LIN {X 0,Y 311.658,Z 464.201,A -85,B 0,C 180,E1 -15739.607,E2 -15739.607} C_VEL
LIN {X 0,Y 311.053,Z 468.336,A -85,B 0,C 180,E1 -15742.209,E2 -15742.209} C_VEL
LIN {X 0,Y 310.773,Z 471.242,A -85,B 0,C 180,E1 -15744.81,E2 -15744.81} C_VEL
LIN {X 0,Y 310.678,Z 472.99,A -85,B 0,C 180,E1 -15747.407,E2 -15747.407} C_VEL
LIN {X 0,Y 310.617,Z 473.6,A -85,B 0,C 180,E1 -15750,E2 -15750} C_VEL
LIN {X 0,Y 310.678,Z 473.032,A -85,B 0,C 180,E1 -15752.593,E2 -15752.593} C_VEL
LIN {X 0,Y 310.76,Z 471.342,A -85,B 0,C 180,E1 -15755.19,E2 -15755.19} C_VEL
LIN {X 0,Y 311.014,Z 468.49,A -85,B 0,C 180,E1 -15757.792,E2 -15757.792} C_VEL
LIN {X 0,Y 311.62,Z 464.406,A -85,B 0,C 180,E1 -15760.395,E2 -15760.395} C_VEL
LIN {X 0,Y 312.631,Z 458.992,A -85,B 0,C 180,E1 -15762.991,E2 -15762.991} C_VEL
LIN {X 0,Y 313.876,Z 452.096,A -85,B 0,C 180,E1 -15765.587,E2 -15765.587} C_VEL
LIN {X 0,Y 315.733,Z 443.488,A -85,B 0,C 180,E1 -15768.158,E2 -15768.158} C_VEL
LIN {X 0,Y 317.704,Z 434.339,A -85,B 0,C 180,E1 -15770.39,E2 -15770.39} C_VEL
LIN {X 0,Y 319.854,Z 424.962,A -85,B 0,C 180,E1 -15772.285,E2 -15772.285} C_VEL
LIN {X 0,Y 322.098,Z 413.952,A -85,B 0,C 180,E1 -15774.149,E2 -15774.149} C_VEL
LIN {X 0,Y 324.511,Z 401.832,A -85,B 0,C 180,E1 -15775.84,E2 -15775.84} C_VEL
LIN {X 0,Y 326.933,Z 388.524,A -85,B 0,C 180,E1 -15777.355,E2 -15777.355} C_VEL
LIN {X 0,Y 329.075,Z 375.209,A -85,B 0,C 180,E1 -15778.572,E2 -15778.572} C_VEL
LIN {X 0,Y 331.025,Z 360.086,A -85,B 0,C 180,E1 -15779.666,E2 -15779.666} C_VEL
LIN {X 0,Y 332.582,Z 345.03,A -85,B 0,C 180,E1 -15780.475,E2 -15780.475} C_VEL
LIN {X 0,Y 333.767,Z 329.274,A -85,B 0,C 180,E1 -15781.057,E2 -15781.057} C_VEL
LIN {X 0,Y 335.921,Z 270.181,A -85,B 0,C 180,E1 -15782.336,E2 -15782.336} C_VEL
LIN {X 0,Y 336.412,Z 254.41,A -85,B 0,C 180,E1 -15782.674,E2 -15782.674} C_VEL
LIN {X 0,Y 336.043,Z 248.619,A -85,B 0,C 180,E1 -15782.859,E2 -15782.859} C_VEL
LIN {X 0,Y 331.98,Z 229.992,A -85,B 0,C 180,E1 -15783.788,E2 -15783.788} C_VEL
LIN {X 0,Y 331.521,Z 224.208,A -85,B 0,C 180,E1 -15783.989,E2 -15783.989} C_VEL
LIN {X 0,Y 331.82,Z 212.788,A -85,B 0,C 180,E1 -15784.246,E2 -15784.246} C_VEL
LIN {X 0,Y 324.4,Z 195.968,A -85,B 0,C 180,E1 -15785.592,E2 -15785.592} C_VEL
LIN {X 0,Y 316.403,Z 180.051,A -85,B 0,C 180,E1 -15787.08,E2 -15787.08} C_VEL
LIN {X 0,Y 308.749,Z 166.539,A -85,B 0,C 180,E1 -15788.556,E2 -15788.556} C_VEL
LIN {X 0,Y 306.876,Z 163.029,A -85,B 0,C 180,E1 -15789.022,E2 -15789.022} C_VEL
LIN {X 0,Y 305.465,Z 158.467,A -85,B 0,C 180,E1 -15790.602,E2 -15790.602} C_VEL
LIN {X 0,Y 305.39,Z 158.081,A -85,B 0,C 180,E1 -15790.91,E2 -15790.91} C_VEL
LIN {X 0,Y 305.399,Z 158.043,A -85,B 0,C 180,E1 -15794.489,E2 -15794.489} C_VEL
LIN {X 0,Y 305.411,Z 158.038,A -85,B 0,C 180,E1 -15798.138,E2 -15798.138} C_VEL
LIN {X 0,Y 305.442,Z 158.029,A -85,B 0,C 180,E1 -15801.592,E2 -15801.592} C_VEL
LIN {X 0,Y 305.463,Z 158.048,A -85,B 0,C 180,E1 -15804.887,E2 -15804.887} C_VEL
LIN {X 0,Y 305.442,Z 158.001,A -85,B 0,C 180,E1 -15808.359,E2 -15808.359} C_VEL
LIN {X 0,Y 305.476,Z 158.046,A -85,B 0,C 180,E1 -15811.109,E2 -15811.109} C_VEL
LIN {X 0,Y 305.482,Z 158.044,A -85,B 0,C 180,E1 -15814.08,E2 -15814.08} C_VEL
LIN {X 0,Y 305.473,Z 158.052,A -85,B 0,C 180,E1 -15818.401,E2 -15818.401} C_VEL
LIN {X 0,Y 305.529,Z 158.052,A -85,B 0,C 180,E1 -15822.6,E2 -15822.6} C_VEL
LIN {X 0,Y 305.625,Z 158.019,A -85,B 0,C 180,E1 -15825.348,E2 -15825.348} C_VEL
LIN {X 0,Y 305.626,Z 158.037,A -85,B 0,C 180,E1 -15829.399,E2 -15829.399} C_VEL
LIN {X 0,Y 305.751,Z 158.004,A -85,B 0,C 180,E1 -15832.073,E2 -15832.073} C_VEL
LIN {X 0,Y 305.669,Z 158.033,A -85,B 0,C 180,E1 -15834.723,E2 -15834.723} C_VEL
LIN {X 0,Y 305.949,Z 157.982,A -85,B 0,C 180,E1 -15838.684,E2 -15838.684} C_VEL
LIN {X 0,Y 305.951,Z 157.995,A -85,B 0,C 180,E1 -15841.316,E2 -15841.316} C_VEL
LIN {X 0,Y 305.671,Z 158.022,A -85,B 0,C 180,E1 -15845.277,E2 -15845.277} C_VEL
LIN {X 0,Y 305.751,Z 158.016,A -85,B 0,C 180,E1 -15847.927,E2 -15847.927} C_VEL
LIN {X 0,Y 305.601,Z 158.043,A -85,B 0,C 180,E1 -15851.945,E2 -15851.945} C_VEL
LIN {X 0,Y 305.639,Z 158.019,A -85,B 0,C 180,E1 -15855.035,E2 -15855.035} C_VEL
LIN {X 0,Y 305.581,Z 158.045,A -85,B 0,C 180,E1 -15858.783,E2 -15858.783} C_VEL
LIN {X 0,Y 305.487,Z 158.055,A -85,B 0,C 180,E1 -15863.039,E2 -15863.039} C_VEL
LIN {X 0,Y 305.527,Z 158.035,A -85,B 0,C 180,E1 -15866.219,E2 -15866.219} C_VEL
LIN {X 0,Y 305.497,Z 158.054,A -85,B 0,C 180,E1 -15869.05,E2 -15869.05} C_VEL
LIN {X 0,Y 305.465,Z 158.001,A -85,B 0,C 180,E1 -15873.517,E2 -15873.517} C_VEL
LIN {X 0,Y 305.473,Z 158.06,A -85,B 0,C 180,E1 -15876.739,E2 -15876.739} C_VEL
LIN {X 0,Y 305.455,Z 158.021,A -85,B 0,C 180,E1 -15880.599,E2 -15880.599} C_VEL
LIN {X 0,Y 305.426,Z 158.066,A -85,B 0,C 180,E1 -15883.655,E2 -15883.655} C_VEL
LIN {X 0,Y 305.506,Z 158.163,A -85,B 0,C 180,E1 -15888.12,E2 -15888.12} C_VEL
LIN {X 0,Y 308.349,Z 167.712,A -85,B 0,C 180,E1 -15891.296,E2 -15891.296} C_VEL
LIN {X 0,Y 316.324,Z 182.462,A -85,B 0,C 180,E1 -15892.89,E2 -15892.89} C_VEL
LIN {X 0,Y 323.257,Z 196.28,A -85,B 0,C 180,E1 -15894.184,E2 -15894.184} C_VEL
LIN {X 0,Y 331.081,Z 213.937,A -85,B 0,C 180,E1 -15895.609,E2 -15895.609} C_VEL
LIN {X 0,Y 331.761,Z 218.64,A -85,B 0,C 180,E1 -15895.81,E2 -15895.81} C_VEL
LIN {X 0,Y 328.229,Z 318.553,A -85,B 0,C 180,E1 -15897.953,E2 -15897.953} C_VEL
LIN {X 0,Y 327.363,Z 337.959,A -85,B 0,C 180,E1 -15898.446,E2 -15898.446} C_VEL
LIN {X 0,Y 325.998,Z 353.359,A -85,B 0,C 180,E1 -15899.067,E2 -15899.067} C_VEL
LIN {X 0,Y 324.342,Z 367.08,A -85,B 0,C 180,E1 -15899.838,E2 -15899.838} C_VEL
LIN {X 0,Y 322.371,Z 381.795,A -85,B 0,C 180,E1 -15900.949,E2 -15900.949} C_VEL
LIN {X 0,Y 320.123,Z 394.944,A -85,B 0,C 180,E1 -15902.191,E2 -15902.191} C_VEL
LIN {X 0,Y 317.506,Z 408.093,A -85,B 0,C 180,E1 -15903.724,E2 -15903.724} C_VEL
LIN {X 0,Y 315.186,Z 419.121,A -85,B 0,C 180,E1 -15905.286,E2 -15905.286} C_VEL
LIN {X 0,Y 312.947,Z 429.414,A -85,B 0,C 180,E1 -15907.037,E2 -15907.037} C_VEL
LIN {X 0,Y 310.691,Z 439.64,A -85,B 0,C 180,E1 -15909.128,E2 -15909.128} C_VEL
LIN {X 0,Y 308.58,Z 448.862,A -85,B 0,C 180,E1 -15911.406,E2 -15911.406} C_VEL
LIN {X 0,Y 306.705,Z 457.543,A -85,B 0,C 180,E1 -15914.039,E2 -15914.039} C_VEL
LIN {X 0,Y 305.38,Z 464.508,A -85,B 0,C 180,E1 -15916.695,E2 -15916.695} C_VEL
LIN {X 0,Y 304.395,Z 469.982,A -85,B 0,C 180,E1 -15919.356,E2 -15919.356} C_VEL
LIN {X 0,Y 303.868,Z 474.121,A -85,B 0,C 180,E1 -15922.023,E2 -15922.023} C_VEL
LIN {X 0,Y 303.596,Z 477.021,A -85,B 0,C 180,E1 -15924.687,E2 -15924.687} C_VEL
LIN {X 0,Y 303.57,Z 478.751,A -85,B 0,C 180,E1 -15927.346,E2 -15927.346} C_VEL
LIN {X 0,Y 303.531,Z 479.341,A -85,B 0,C 180,E1 -15930,E2 -15930} C_VEL
LIN {X 0,Y 303.57,Z 478.741,A -85,B 0,C 180,E1 -15932.654,E2 -15932.654} C_VEL
LIN {X 0,Y 303.624,Z 476.802,A -85,B 0,C 180,E1 -15935.544,E2 -15935.544} C_VEL
LIN {X 0,Y 303.867,Z 474.09,A -85,B 0,C 180,E1 -15937.977,E2 -15937.977} C_VEL
LIN {X 0,Y 304.388,Z 469.945,A -85,B 0,C 180,E1 -15940.644,E2 -15940.644} C_VEL
LIN {X 0,Y 305.369,Z 464.455,A -85,B 0,C 180,E1 -15943.306,E2 -15943.306} C_VEL
LIN {X 0,Y 306.657,Z 457.468,A -85,B 0,C 180,E1 -15945.963,E2 -15945.963} C_VEL
LIN {X 0,Y 308.568,Z 448.775,A -85,B 0,C 180,E1 -15948.594,E2 -15948.594} C_VEL
LIN {X 0,Y 310.704,Z 439.539,A -85,B 0,C 180,E1 -15950.871,E2 -15950.871} C_VEL
LIN {X 0,Y 312.746,Z 429.81,A -85,B 0,C 180,E1 -15952.876,E2 -15952.876} C_VEL
LIN {X 0,Y 315.433,Z 417.964,A -85,B 0,C 180,E1 -15954.869,E2 -15954.869} C_VEL
LIN {X 0,Y 317.982,Z 405.536,A -85,B 0,C 180,E1 -15956.587,E2 -15956.587} C_VEL
LIN {X 0,Y 320.353,Z 393.309,A -85,B 0,C 180,E1 -15957.965,E2 -15957.965} C_VEL
LIN {X 0,Y 322.79,Z 378.654,A -85,B 0,C 180,E1 -15959.297,E2 -15959.297} C_VEL
LIN {X 0,Y 324.654,Z 364.495,A -85,B 0,C 180,E1 -15960.309,E2 -15960.309} C_VEL
LIN {X 0,Y 326.377,Z 349.088,A -85,B 0,C 180,E1 -15961.118,E2 -15961.118} C_VEL
LIN {X 0,Y 327.591,Z 333.851,A -85,B 0,C 180,E1 -15961.664,E2 -15961.664} C_VEL
LIN {X 0,Y 331.459,Z 224.627,A -85,B 0,C 180,E1 -15964.044,E2 -15964.044} C_VEL
LIN {X 0,Y 331.527,Z 216.912,A -85,B 0,C 180,E1 -15964.233,E2 -15964.233} C_VEL
LIN {X 0,Y 330.749,Z 213.239,A -85,B 0,C 180,E1 -15964.419,E2 -15964.419} C_VEL
LIN {X 0,Y 322.793,Z 195.303,A -85,B 0,C 180,E1 -15965.87,E2 -15965.87} C_VEL
LIN {X 0,Y 314.623,Z 179.237,A -85,B 0,C 180,E1 -15967.4,E2 -15967.4} C_VEL
LIN {X 0,Y 309.575,Z 170.227,A -85,B 0,C 180,E1 -15968.376,E2 -15968.376} C_VEL
LIN {X 0,Y 308.28,Z 167.558,A -85,B 0,C 180,E1 -15968.701,E2 -15968.701} C_VEL
LIN {X 0,Y 305.477,Z 158.164,A -85,B 0,C 180,E1 -15971.851,E2 -15971.851} C_VEL
LIN {X 0,Y 305.4,Z 158.054,A -85,B 0,C 180,E1 -15975.511,E2 -15975.511} C_VEL
LIN {X 0,Y 305.44,Z 158.034,A -85,B 0,C 180,E1 -15978.143,E2 -15978.143} C_VEL
LIN {X 0,Y 305.495,Z 158.041,A -85,B 0,C 180,E1 -15981.6,E2 -15981.6} C_VEL
LIN {X 0,Y 305.462,Z 158.025,A -85,B 0,C 180,E1 -15984.887,E2 -15984.887} C_VEL
LIN {X 0,Y 305.451,Z 158.011,A -85,B 0,C 180,E1 -15988.355,E2 -15988.355} C_VEL
LIN {X 0,Y 305.521,Z 158.053,A -85,B 0,C 180,E1 -15991.114,E2 -15991.114} C_VEL
LIN {X 0,Y 305.572,Z 158.029,A -85,B 0,C 180,E1 -15994.088,E2 -15994.088} C_VEL
LIN {X 0,Y 305.501,Z 158.039,A -85,B 0,C 180,E1 -15998.403,E2 -15998.403} C_VEL
LIN {X 0,Y 305.591,Z 158.044,A -85,B 0,C 180,E1 -16001.218,E2 -16001.218} C_VEL
LIN {X 0,Y 305.65,Z 158.021,A -85,B 0,C 180,E1 -16005.349,E2 -16005.349} C_VEL
LIN {X 0,Y 305.625,Z 158.022,A -85,B 0,C 180,E1 -16009.399,E2 -16009.399} C_VEL
LIN {X 0,Y 305.75,Z 158.016,A -85,B 0,C 180,E1 -16012.073,E2 -16012.073} C_VEL
LIN {X 0,Y 305.671,Z 158.022,A -85,B 0,C 180,E1 -16014.723,E2 -16014.723} C_VEL
LIN {X 0,Y 305.953,Z 157.994,A -85,B 0,C 180,E1 -16018.684,E2 -16018.684} C_VEL
LIN {X 0,Y 305.951,Z 157.982,A -85,B 0,C 180,E1 -16021.316,E2 -16021.316} C_VEL
LIN {X 0,Y 305.794,Z 158.012,A -85,B 0,C 180,E1 -16026.599,E2 -16026.599} C_VEL
LIN {X 0,Y 305.695,Z 158.012,A -85,B 0,C 180,E1 -16029.261,E2 -16029.261} C_VEL
LIN {X 0,Y 305.587,Z 158.031,A -85,B 0,C 180,E1 -16033.296,E2 -16033.296} C_VEL
LIN {X 0,Y 305.552,Z 158.039,A -85,B 0,C 180,E1 -16036.023,E2 -16036.023} C_VEL
LIN {X 0,Y 305.484,Z 158.038,A -85,B 0,C 180,E1 -16040.188,E2 -16040.188} C_VEL
LIN {X 0,Y 305.442,Z 158.048,A -85,B 0,C 180,E1 -16044.467,E2 -16044.467} C_VEL
LIN {X 0,Y 305.452,Z 158.061,A -85,B 0,C 180,E1 -16047.398,E2 -16047.398} C_VEL
LIN {X 0,Y 305.429,Z 158.02,A -85,B 0,C 180,E1 -16050.413,E2 -16050.413} C_VEL
LIN {X 0,Y 305.465,Z 158.017,A -85,B 0,C 180,E1 -16054.078,E2 -16054.078} C_VEL
LIN {X 0,Y 305.469,Z 158.062,A -85,B 0,C 180,E1 -16056.74,E2 -16056.74} C_VEL
LIN {X 0,Y 305.409,Z 158.019,A -85,B 0,C 180,E1 -16060.59,E2 -16060.59} C_VEL
LIN {X 0,Y 305.421,Z 158.066,A -85,B 0,C 180,E1 -16063.656,E2 -16063.656} C_VEL
LIN {X 0,Y 305.435,Z 158.05,A -85,B 0,C 180,E1 -16067.419,E2 -16067.419} C_VEL
LIN {X 0,Y 305.42,Z 158.229,A -85,B 0,C 180,E1 -16069.408,E2 -16069.408} C_VEL
LIN {X 0,Y 306.99,Z 163.275,A -85,B 0,C 180,E1 -16071.167,E2 -16071.167} C_VEL
LIN {X 0,Y 314.485,Z 176.51,A -85,B 0,C 180,E1 -16072.68,E2 -16072.68} C_VEL
LIN {X 0,Y 322.078,Z 191.253,A -85,B 0,C 180,E1 -16074.106,E2 -16074.106} C_VEL
LIN {X 0,Y 329.975,Z 208.394,A -85,B 0,C 180,E1 -16075.54,E2 -16075.54} C_VEL
LIN {X 0,Y 331.749,Z 212.616,A -85,B 0,C 180,E1 -16075.859,E2 -16075.859} C_VEL
LIN {X 0,Y 328.421,Z 312.293,A -85,B 0,C 180,E1 -16078.019,E2 -16078.019} C_VEL
LIN {X 0,Y 327.446,Z 332.079,A -85,B 0,C 180,E1 -16078.5,E2 -16078.5} C_VEL
LIN {X 0,Y 326.21,Z 347.317,A -85,B 0,C 180,E1 -16079.112,E2 -16079.112} C_VEL
LIN {X 0,Y 324.689,Z 361.386,A -85,B 0,C 180,E1 -16079.909,E2 -16079.909} C_VEL
LIN {X 0,Y 322.785,Z 375.372,A -85,B 0,C 180,E1 -16080.946,E2 -16080.946} C_VEL
LIN {X 0,Y 320.494,Z 389.08,A -85,B 0,C 180,E1 -16082.226,E2 -16082.226} C_VEL
LIN {X 0,Y 318.241,Z 401.138,A -85,B 0,C 180,E1 -16083.613,E2 -16083.613} C_VEL
LIN {X 0,Y 315.637,Z 413.38,A -85,B 0,C 180,E1 -16085.324,E2 -16085.324} C_VEL
LIN {X 0,Y 313.181,Z 425.143,A -85,B 0,C 180,E1 -16087.354,E2 -16087.354} C_VEL
LIN {X 0,Y 310.79,Z 435.369,A -85,B 0,C 180,E1 -16089.482,E2 -16089.482} C_VEL
LIN {X 0,Y 308.73,Z 444.365,A -85,B 0,C 180,E1 -16091.759,E2 -16091.759} C_VEL
LIN {X 0,Y 306.988,Z 451.821,A -85,B 0,C 180,E1 -16094.055,E2 -16094.055} C_VEL
LIN {X 0,Y 305.697,Z 458.79,A -85,B 0,C 180,E1 -16096.709,E2 -16096.709} C_VEL
LIN {X 0,Y 304.634,Z 464.268,A -85,B 0,C 180,E1 -16099.364,E2 -16099.364} C_VEL
LIN {X 0,Y 304.006,Z 468.404,A -85,B 0,C 180,E1 -16102.027,E2 -16102.027} C_VEL
LIN {X 0,Y 303.686,Z 471.309,A -85,B 0,C 180,E1 -16104.689,E2 -16104.689} C_VEL
LIN {X 0,Y 303.604,Z 473.056,A -85,B 0,C 180,E1 -16107.346,E2 -16107.346} C_VEL
LIN {X 0,Y 303.533,Z 473.666,A -85,B 0,C 180,E1 -16110,E2 -16110} C_VEL
LIN {X 0,Y 303.603,Z 473.098,A -85,B 0,C 180,E1 -16112.654,E2 -16112.654} C_VEL
LIN {X 0,Y 303.73,Z 471.045,A -85,B 0,C 180,E1 -16115.744,E2 -16115.744} C_VEL
LIN {X 0,Y 303.976,Z 468.555,A -85,B 0,C 180,E1 -16117.974,E2 -16117.974} C_VEL
LIN {X 0,Y 304.602,Z 464.471,A -85,B 0,C 180,E1 -16120.637,E2 -16120.637} C_VEL
LIN {X 0,Y 305.657,Z 459.057,A -85,B 0,C 180,E1 -16123.293,E2 -16123.293} C_VEL
LIN {X 0,Y 306.989,Z 452.161,A -85,B 0,C 180,E1 -16125.945,E2 -16125.945} C_VEL
LIN {X 0,Y 308.94,Z 443.553,A -85,B 0,C 180,E1 -16128.571,E2 -16128.571} C_VEL
LIN {X 0,Y 311.026,Z 434.403,A -85,B 0,C 180,E1 -16130.848,E2 -16130.848} C_VEL
LIN {X 0,Y 313.174,Z 425.31,A -85,B 0,C 180,E1 -16132.726,E2 -16132.726} C_VEL
LIN {X 0,Y 315.592,Z 414.015,A -85,B 0,C 180,E1 -16134.68,E2 -16134.68} C_VEL
LIN {X 0,Y 318.088,Z 401.895,A -85,B 0,C 180,E1 -16136.401,E2 -16136.401} C_VEL
LIN {X 0,Y 320.625,Z 388.586,A -85,B 0,C 180,E1 -16137.939,E2 -16137.939} C_VEL
LIN {X 0,Y 322.811,Z 375.586,A -85,B 0,C 180,E1 -16139.147,E2 -16139.147} C_VEL
LIN {X 0,Y 324.731,Z 361.274,A -85,B 0,C 180,E1 -16140.211,E2 -16140.211} C_VEL
LIN {X 0,Y 326.352,Z 346.609,A -85,B 0,C 180,E1 -16141.031,E2 -16141.031} C_VEL
LIN {X 0,Y 327.575,Z 331.603,A -85,B 0,C 180,E1 -16141.621,E2 -16141.621} C_VEL
LIN {X 0,Y 328.533,Z 309.767,A -85,B 0,C 180,E1 -16142.149,E2 -16142.149} C_VEL
LIN {X 0,Y 331.521,Z 224.208,A -85,B 0,C 180,E1 -16143.989,E2 -16143.989} C_VEL
LIN {X 0,Y 330.934,Z 220.467,A -85,B 0,C 180,E1 -16144.153,E2 -16144.153} C_VEL
LIN {X 0,Y 329.477,Z 217.097,A -85,B 0,C 180,E1 -16144.413,E2 -16144.413} C_VEL
LIN {X 0,Y 322.573,Z 206.994,A -85,B 0,C 180,E1 -16145.529,E2 -16145.529} C_VEL
LIN {X 0,Y 314.231,Z 189.381,A -85,B 0,C 180,E1 -16147.118,E2 -16147.118} C_VEL
LIN {X 0,Y 306.471,Z 175.095,A -85,B 0,C 180,E1 -16148.644,E2 -16148.644} C_VEL
LIN {X 0,Y 299.708,Z 163.412,A -85,B 0,C 180,E1 -16150.089,E2 -16150.089} C_VEL
LIN {X 0,Y 298.405,Z 159.201,A -85,B 0,C 180,E1 -16151.593,E2 -16151.593} C_VEL
LIN {X 0,Y 298.37,Z 158.924,A -85,B 0,C 180,E1 -16153.097,E2 -16153.097} C_VEL
LIN {X 0,Y 298.371,Z 158.944,A -85,B 0,C 180,E1 -16156.915,E2 -16156.915} C_VEL
LIN {X 0,Y 298.352,Z 158.902,A -85,B 0,C 180,E1 -16161.019,E2 -16161.019} C_VEL
LIN {X 0,Y 298.406,Z 158.942,A -85,B 0,C 180,E1 -16163.928,E2 -16163.928} C_VEL
LIN {X 0,Y 298.393,Z 158.88,A -85,B 0,C 180,E1 -16167.199,E2 -16167.199} C_VEL
LIN {X 0,Y 298.402,Z 158.917,A -85,B 0,C 180,E1 -16170.625,E2 -16170.625} C_VEL
LIN {X 0,Y 298.416,Z 158.92,A -85,B 0,C 180,E1 -16174.918,E2 -16174.918} C_VEL
LIN {X 0,Y 298.401,Z 158.939,A -85,B 0,C 180,E1 -16177.862,E2 -16177.862} C_VEL
LIN {X 0,Y 298.465,Z 158.914,A -85,B 0,C 180,E1 -16180.752,E2 -16180.752} C_VEL
LIN {X 0,Y 298.587,Z 158.897,A -85,B 0,C 180,E1 -16184.994,E2 -16184.994} C_VEL
LIN {X 0,Y 298.585,Z 158.917,A -85,B 0,C 180,E1 -16189.146,E2 -16189.146} C_VEL
LIN {X 0,Y 298.702,Z 158.88,A -85,B 0,C 180,E1 -16191.884,E2 -16191.884} C_VEL
LIN {X 0,Y 298.639,Z 158.909,A -85,B 0,C 180,E1 -16194.598,E2 -16194.598} C_VEL
LIN {X 0,Y 298.916,Z 158.857,A -85,B 0,C 180,E1 -16198.653,E2 -16198.653} C_VEL
LIN {X 0,Y 298.918,Z 158.87,A -85,B 0,C 180,E1 -16201.347,E2 -16201.347} C_VEL
LIN {X 0,Y 298.64,Z 158.899,A -85,B 0,C 180,E1 -16205.401,E2 -16205.401} C_VEL
LIN {X 0,Y 298.702,Z 158.892,A -85,B 0,C 180,E1 -16208.115,E2 -16208.115} C_VEL
LIN {X 0,Y 298.553,Z 158.92,A -85,B 0,C 180,E1 -16212.231,E2 -16212.231} C_VEL
LIN {X 0,Y 298.607,Z 158.894,A -85,B 0,C 180,E1 -16215.209,E2 -16215.209} C_VEL
LIN {X 0,Y 298.527,Z 158.919,A -85,B 0,C 180,E1 -16219.244,E2 -16219.244} C_VEL
LIN {X 0,Y 298.43,Z 158.936,A -85,B 0,C 180,E1 -16223.6,E2 -16223.6} C_VEL
LIN {X 0,Y 298.487,Z 158.912,A -85,B 0,C 180,E1 -16226.574,E2 -16226.574} C_VEL
LIN {X 0,Y 298.422,Z 158.927,A -85,B 0,C 180,E1 -16229.641,E2 -16229.641} C_VEL
LIN {X 0,Y 298.396,Z 158.878,A -85,B 0,C 180,E1 -16232.8,E2 -16232.8} C_VEL
LIN {X 0,Y 298.445,Z 158.936,A -85,B 0,C 180,E1 -16236.807,E2 -16236.807} C_VEL
LIN {X 0,Y 298.387,Z 158.903,A -85,B 0,C 180,E1 -16241.087,E2 -16241.087} C_VEL
LIN {X 0,Y 298.399,Z 158.939,A -85,B 0,C 180,E1 -16243.103,E2 -16243.103} C_VEL
LIN {X 0,Y 298.447,Z 159.078,A -85,B 0,C 180,E1 -16247.211,E2 -16247.211} C_VEL
LIN {X 0,Y 301.023,Z 167.6,A -85,B 0,C 180,E1 -16250.165,E2 -16250.165} C_VEL
LIN {X 0,Y 308.862,Z 181.664,A -85,B 0,C 180,E1 -16251.814,E2 -16251.814} C_VEL
LIN {X 0,Y 316.721,Z 197.093,A -85,B 0,C 180,E1 -16253.35,E2 -16253.35} C_VEL
LIN {X 0,Y 324.301,Z 213.884,A -85,B 0,C 180,E1 -16254.785,E2 -16254.785} C_VEL
LIN {X 0,Y 325.615,Z 217.399,A -85,B 0,C 180,E1 -16255.041,E2 -16255.041} C_VEL
LIN {X 0,Y 325.839,Z 220.532,A -85,B 0,C 180,E1 -16255.151,E2 -16255.151} C_VEL
LIN {X 0,Y 321.658,Z 333.25,A -85,B 0,C 180,E1 -16257.635,E2 -16257.635} C_VEL
LIN {X 0,Y 320.42,Z 348.658,A -85,B 0,C 180,E1 -16258.19,E2 -16258.19} C_VEL
LIN {X 0,Y 318.687,Z 363.552,A -85,B 0,C 180,E1 -16258.97,E2 -16258.97} C_VEL
LIN {X 0,Y 316.849,Z 377.218,A -85,B 0,C 180,E1 -16259.943,E2 -16259.943} C_VEL
LIN {X 0,Y 314.643,Z 390.368,A -85,B 0,C 180,E1 -16261.117,E2 -16261.117} C_VEL
LIN {X 0,Y 312.16,Z 403.064,A -85,B 0,C 180,E1 -16262.513,E2 -16262.513} C_VEL
LIN {X 0,Y 309.452,Z 415.905,A -85,B 0,C 180,E1 -16264.256,E2 -16264.256} C_VEL
LIN {X 0,Y 307.023,Z 426.604,A -85,B 0,C 180,E1 -16266.016,E2 -16266.016} C_VEL
LIN {X 0,Y 304.739,Z 436.601,A -85,B 0,C 180,E1 -16267.99,E2 -16267.99} C_VEL
LIN {X 0,Y 302.377,Z 446.329,A -85,B 0,C 180,E1 -16270.305,E2 -16270.305} C_VEL
LIN {X 0,Y 300.448,Z 454.446,A -85,B 0,C 180,E1 -16272.648,E2 -16272.648} C_VEL
LIN {X 0,Y 299.056,Z 461.158,A -85,B 0,C 180,E1 -16275.018,E2 -16275.018} C_VEL
LIN {X 0,Y 297.799,Z 467.354,A -85,B 0,C 180,E1 -16277.737,E2 -16277.737} C_VEL
LIN {X 0,Y 297.052,Z 472.145,A -85,B 0,C 180,E1 -16280.467,E2 -16280.467} C_VEL
LIN {X 0,Y 296.642,Z 475.655,A -85,B 0,C 180,E1 -16283.197,E2 -16283.197} C_VEL
LIN {X 0,Y 296.468,Z 477.963,A -85,B 0,C 180,E1 -16285.922,E2 -16285.922} C_VEL
LIN {X 0,Y 296.444,Z 479.123,A -85,B 0,C 180,E1 -16288.641,E2 -16288.641} C_VEL
LIN {X 0,Y 296.444,Z 479.119,A -85,B 0,C 180,E1 -16291.358,E2 -16291.358} C_VEL
LIN {X 0,Y 296.469,Z 477.946,A -85,B 0,C 180,E1 -16294.078,E2 -16294.078} C_VEL
LIN {X 0,Y 296.642,Z 475.626,A -85,B 0,C 180,E1 -16296.803,E2 -16296.803} C_VEL
LIN {X 0,Y 297.048,Z 472.11,A -85,B 0,C 180,E1 -16299.533,E2 -16299.533} C_VEL
LIN {X 0,Y 297.795,Z 467.309,A -85,B 0,C 180,E1 -16302.263,E2 -16302.263} C_VEL
LIN {X 0,Y 299.009,Z 461.091,A -85,B 0,C 180,E1 -16304.984,E2 -16304.984} C_VEL
LIN {X 0,Y 300.715,Z 453.283,A -85,B 0,C 180,E1 -16307.687,E2 -16307.687} C_VEL
LIN {X 0,Y 302.622,Z 444.979,A -85,B 0,C 180,E1 -16310.032,E2 -16310.032} C_VEL
LIN {X 0,Y 305.081,Z 434.973,A -85,B 0,C 180,E1 -16312.34,E2 -16312.34} C_VEL
LIN {X 0,Y 306.924,Z 426.703,A -85,B 0,C 180,E1 -16313.946,E2 -16313.946} C_VEL
LIN {X 0,Y 309.459,Z 415.754,A -85,B 0,C 180,E1 -16315.743,E2 -16315.743} C_VEL
LIN {X 0,Y 311.903,Z 404.172,A -85,B 0,C 180,E1 -16317.329,E2 -16317.329} C_VEL
LIN {X 0,Y 314.338,Z 391.709,A -85,B 0,C 180,E1 -16318.731,E2 -16318.731} C_VEL
LIN {X 0,Y 316.759,Z 377.497,A -85,B 0,C 180,E1 -16320.012,E2 -16320.012} C_VEL
LIN {X 0,Y 318.667,Z 363.166,A -85,B 0,C 180,E1 -16321.032,E2 -16321.032} C_VEL
LIN {X 0,Y 320.406,Z 348.118,A -85,B 0,C 180,E1 -16321.811,E2 -16321.811} C_VEL
LIN {X 0,Y 321.585,Z 333.77,A -85,B 0,C 180,E1 -16322.327,E2 -16322.327} C_VEL
LIN {X 0,Y 325.684,Z 222.129,A -85,B 0,C 180,E1 -16324.796,E2 -16324.796} C_VEL
LIN {X 0,Y 325.534,Z 217.472,A -85,B 0,C 180,E1 -16324.937,E2 -16324.937} C_VEL
LIN {X 0,Y 323.681,Z 212.486,A -85,B 0,C 180,E1 -16325.298,E2 -16325.298} C_VEL
LIN {X 0,Y 315.367,Z 194.343,A -85,B 0,C 180,E1 -16326.875,E2 -16326.875} C_VEL
LIN {X 0,Y 307.59,Z 179.407,A -85,B 0,C 180,E1 -16328.4,E2 -16328.4} C_VEL
LIN {X 0,Y 301.013,Z 167.567,A -85,B 0,C 180,E1 -16329.8,E2 -16329.8} C_VEL
LIN {X 0,Y 298.452,Z 159.06,A -85,B 0,C 180,E1 -16332.756,E2 -16332.756} C_VEL
LIN {X 0,Y 298.403,Z 158.936,A -85,B 0,C 180,E1 -16336.921,E2 -16336.921} C_VEL
LIN {X 0,Y 298.415,Z 158.909,A -85,B 0,C 180,E1 -16341.004,E2 -16341.004} C_VEL
LIN {X 0,Y 298.432,Z 158.924,A -85,B 0,C 180,E1 -16343.932,E2 -16343.932} C_VEL
LIN {X 0,Y 298.395,Z 158.883,A -85,B 0,C 180,E1 -16347.984,E2 -16347.984} C_VEL
LIN {X 0,Y 298.464,Z 158.931,A -85,B 0,C 180,E1 -16351.905,E2 -16351.905} C_VEL
LIN {X 0,Y 298.487,Z 158.918,A -85,B 0,C 180,E1 -16354.924,E2 -16354.924} C_VEL
LIN {X 0,Y 298.45,Z 158.915,A -85,B 0,C 180,E1 -16359.315,E2 -16359.315} C_VEL
LIN {X 0,Y 298.539,Z 158.922,A -85,B 0,C 180,E1 -16362.18,E2 -16362.18} C_VEL
LIN {X 0,Y 298.594,Z 158.896,A -85,B 0,C 180,E1 -16364.995,E2 -16364.995} C_VEL
LIN {X 0,Y 298.584,Z 158.902,A -85,B 0,C 180,E1 -16369.146,E2 -16369.146} C_VEL
LIN {X 0,Y 298.701,Z 158.892,A -85,B 0,C 180,E1 -16371.885,E2 -16371.885} C_VEL
LIN {X 0,Y 298.64,Z 158.899,A -85,B 0,C 180,E1 -16374.599,E2 -16374.599} C_VEL
LIN {X 0,Y 298.92,Z 158.869,A -85,B 0,C 180,E1 -16378.653,E2 -16378.653} C_VEL
LIN {X 0,Y 298.917,Z 158.857,A -85,B 0,C 180,E1 -16381.347,E2 -16381.347} C_VEL
LIN {X 0,Y 298.742,Z 158.889,A -85,B 0,C 180,E1 -16386.755,E2 -16386.755} C_VEL
LIN {X 0,Y 298.626,Z 158.894,A -85,B 0,C 180,E1 -16389.482,E2 -16389.482} C_VEL
LIN {X 0,Y 298.546,Z 158.904,A -85,B 0,C 180,E1 -16393.616,E2 -16393.616} C_VEL
LIN {X 0,Y 298.485,Z 158.924,A -85,B 0,C 180,E1 -16396.412,E2 -16396.412} C_VEL
LIN {X 0,Y 298.443,Z 158.916,A -85,B 0,C 180,E1 -16399.617,E2 -16399.617} C_VEL
LIN {X 0,Y 298.383,Z 158.936,A -85,B 0,C 180,E1 -16403.604,E2 -16403.604} C_VEL
LIN {X 0,Y 298.403,Z 158.932,A -85,B 0,C 180,E1 -16406.583,E2 -16406.583} C_VEL
LIN {X 0,Y 298.393,Z 158.914,A -85,B 0,C 180,E1 -16409.644,E2 -16409.644} C_VEL
LIN {X 0,Y 298.393,Z 158.878,A -85,B 0,C 180,E1 -16412.801,E2 -16412.801} C_VEL
LIN {X 0,Y 298.441,Z 158.936,A -85,B 0,C 180,E1 -16416.806,E2 -16416.806} C_VEL
LIN {X 0,Y 298.347,Z 158.904,A -85,B 0,C 180,E1 -16421.268,E2 -16421.268} C_VEL
LIN {X 0,Y 298.355,Z 158.925,A -85,B 0,C 180,E1 -16425.035,E2 -16425.035} C_VEL
LIN {X 0,Y 298.384,Z 159.148,A -85,B 0,C 180,E1 -16428.513,E2 -16428.513} C_VEL
LIN {X 0,Y 299.702,Z 163.418,A -85,B 0,C 180,E1 -16430.041,E2 -16430.041} C_VEL
LIN {X 0,Y 307.751,Z 177.282,A -85,B 0,C 180,E1 -16431.738,E2 -16431.738} C_VEL
LIN {X 0,Y 315.801,Z 192.661,A -85,B 0,C 180,E1 -16433.313,E2 -16433.313} C_VEL
LIN {X 0,Y 322.916,Z 207.888,A -85,B 0,C 180,E1 -16434.659,E2 -16434.659} C_VEL
LIN {X 0,Y 325.822,Z 214.611,A -85,B 0,C 180,E1 -16435.199,E2 -16435.199} C_VEL
LIN {X 0,Y 322.71,Z 303.444,A -85,B 0,C 180,E1 -16437.152,E2 -16437.152} C_VEL
LIN {X 0,Y 321.636,Z 329.879,A -85,B 0,C 180,E1 -16437.772,E2 -16437.772} C_VEL
LIN {X 0,Y 320.424,Z 344.728,A -85,B 0,C 180,E1 -16438.33,E2 -16438.33} C_VEL
LIN {X 0,Y 318.745,Z 359.891,A -85,B 0,C 180,E1 -16439.16,E2 -16439.16} C_VEL
LIN {X 0,Y 316.764,Z 374.379,A -85,B 0,C 180,E1 -16440.228,E2 -16440.228} C_VEL
LIN {X 0,Y 314.51,Z 387.721,A -85,B 0,C 180,E1 -16441.468,E2 -16441.468} C_VEL
LIN {X 0,Y 311.858,Z 401.208,A -85,B 0,C 180,E1 -16443.029,E2 -16443.029} C_VEL
LIN {X 0,Y 309.172,Z 413.45,A -85,B 0,C 180,E1 -16444.772,E2 -16444.772} C_VEL
LIN {X 0,Y 306.702,Z 424.754,A -85,B 0,C 180,E1 -16446.748,E2 -16446.748} C_VEL
LIN {X 0,Y 304.099,Z 435.438,A -85,B 0,C 180,E1 -16449.009,E2 -16449.009} C_VEL
LIN {X 0,Y 301.961,Z 444.434,A -85,B 0,C 180,E1 -16451.336,E2 -16451.336} C_VEL
LIN {X 0,Y 300.012,Z 452.349,A -85,B 0,C 180,E1 -16453.833,E2 -16453.833} C_VEL
LIN {X 0,Y 298.741,Z 458.858,A -85,B 0,C 180,E1 -16456.393,E2 -16456.393} C_VEL
LIN {X 0,Y 297.621,Z 464.336,A -85,B 0,C 180,E1 -16459.111,E2 -16459.111} C_VEL
LIN {X 0,Y 296.951,Z 468.471,A -85,B 0,C 180,E1 -16461.836,E2 -16461.836} C_VEL
LIN {X 0,Y 296.621,Z 471.376,A -85,B 0,C 180,E1 -16464.562,E2 -16464.562} C_VEL
LIN {X 0,Y 296.531,Z 473.122,A -85,B 0,C 180,E1 -16467.283,E2 -16467.283} C_VEL
LIN {X 0,Y 296.452,Z 473.732,A -85,B 0,C 180,E1 -16470,E2 -16470} C_VEL
LIN {X 0,Y 296.53,Z 473.164,A -85,B 0,C 180,E1 -16472.717,E2 -16472.717} C_VEL
LIN {X 0,Y 296.631,Z 471.279,A -85,B 0,C 180,E1 -16475.676,E2 -16475.676} C_VEL
LIN {X 0,Y 296.928,Z 468.621,A -85,B 0,C 180,E1 -16478.165,E2 -16478.165} C_VEL
LIN {X 0,Y 297.594,Z 464.537,A -85,B 0,C 180,E1 -16480.89,E2 -16480.89} C_VEL
LIN {X 0,Y 298.699,Z 459.123,A -85,B 0,C 180,E1 -16483.609,E2 -16483.609} C_VEL
LIN {X 0,Y 300.118,Z 452.226,A -85,B 0,C 180,E1 -16486.321,E2 -16486.321} C_VEL
LIN {X 0,Y 302.17,Z 443.618,A -85,B 0,C 180,E1 -16489.003,E2 -16489.003} C_VEL
LIN {X 0,Y 304.356,Z 434.468,A -85,B 0,C 180,E1 -16491.327,E2 -16491.327} C_VEL
LIN {X 0,Y 306.521,Z 425.637,A -85,B 0,C 180,E1 -16493.19,E2 -16493.19} C_VEL
LIN {X 0,Y 309.138,Z 414.079,A -85,B 0,C 180,E1 -16495.231,E2 -16495.231} C_VEL
LIN {X 0,Y 311.728,Z 401.957,A -85,B 0,C 180,E1 -16496.983,E2 -16496.983} C_VEL
LIN {X 0,Y 314.362,Z 388.648,A -85,B 0,C 180,E1 -16498.546,E2 -16498.546} C_VEL
LIN {X 0,Y 316.717,Z 375.07,A -85,B 0,C 180,E1 -16499.824,E2 -16499.824} C_VEL
LIN {X 0,Y 318.739,Z 360.204,A -85,B 0,C 180,E1 -16500.933,E2 -16500.933} C_VEL
LIN {X 0,Y 320.431,Z 345.142,A -85,B 0,C 180,E1 -16501.762,E2 -16501.762} C_VEL
LIN {X 0,Y 321.691,Z 329.375,A -85,B 0,C 180,E1 -16502.361,E2 -16502.361} C_VEL
LIN {X 0,Y 324.144,Z 267.714,A -85,B 0,C 180,E1 -16503.73,E2 -16503.73} C_VEL
LIN {X 0,Y 325.898,Z 214.764,A -85,B 0,C 180,E1 -16504.907,E2 -16504.907} C_VEL
LIN {X 0,Y 322.573,Z 206.994,A -85,B 0,C 180,E1 -16505.529,E2 -16505.529} C_VEL
LIN {X 0,Y 318.53,Z 201.352,A -85,B 0,C 180,E1 -16506.205,E2 -16506.205} C_VEL
LIN {X 0,Y 309.29,Z 191.562,A -85,B 0,C 180,E1 -16507.752,E2 -16507.752} C_VEL
LIN {X 0,Y 305.39,Z 185.929,A -85,B 0,C 180,E1 -16508.487,E2 -16508.487} C_VEL
LIN {X 0,Y 299.104,Z 174.784,A -85,B 0,C 180,E1 -16509.793,E2 -16509.793} C_VEL
LIN {X 0,Y 292.435,Z 163.633,A -85,B 0,C 180,E1 -16511.282,E2 -16511.282} C_VEL
LIN {X 0,Y 291.354,Z 159.981,A -85,B 0,C 180,E1 -16512.612,E2 -16512.612} C_VEL
LIN {X 0,Y 291.29,Z 159.826,A -85,B 0,C 180,E1 -16516.37,E2 -16516.37} C_VEL
LIN {X 0,Y 291.311,Z 159.774,A -85,B 0,C 180,E1 -16520.535,E2 -16520.535} C_VEL
LIN {X 0,Y 291.397,Z 159.806,A -85,B 0,C 180,E1 -16522.918,E2 -16522.918} C_VEL
LIN {X 0,Y 291.345,Z 159.768,A -85,B 0,C 180,E1 -16526.301,E2 -16526.301} C_VEL
LIN {X 0,Y 291.365,Z 159.781,A -85,B 0,C 180,E1 -16530.268,E2 -16530.268} C_VEL
LIN {X 0,Y 291.344,Z 159.802,A -85,B 0,C 180,E1 -16534.265,E2 -16534.265} C_VEL
LIN {X 0,Y 291.354,Z 159.817,A -85,B 0,C 180,E1 -16537.297,E2 -16537.297} C_VEL
LIN {X 0,Y 291.391,Z 159.793,A -85,B 0,C 180,E1 -16540.265,E2 -16540.265} C_VEL
LIN {X 0,Y 291.499,Z 159.782,A -85,B 0,C 180,E1 -16544.666,E2 -16544.666} C_VEL
LIN {X 0,Y 291.531,Z 159.795,A -85,B 0,C 180,E1 -16548.88,E2 -16548.88} C_VEL
LIN {X 0,Y 291.655,Z 159.757,A -85,B 0,C 180,E1 -16551.687,E2 -16551.687} C_VEL
LIN {X 0,Y 291.608,Z 159.785,A -85,B 0,C 180,E1 -16554.468,E2 -16554.468} C_VEL
LIN {X 0,Y 291.882,Z 159.732,A -85,B 0,C 180,E1 -16558.62,E2 -16558.62} C_VEL
LIN {X 0,Y 291.885,Z 159.745,A -85,B 0,C 180,E1 -16561.38,E2 -16561.38} C_VEL
LIN {X 0,Y 291.693,Z 159.775,A -85,B 0,C 180,E1 -16566.919,E2 -16566.919} C_VEL
LIN {X 0,Y 291.57,Z 159.767,A -85,B 0,C 180,E1 -16569.714,E2 -16569.714} C_VEL
LIN {X 0,Y 291.524,Z 159.788,A -85,B 0,C 180,E1 -16573.95,E2 -16573.95} C_VEL
LIN {X 0,Y 291.488,Z 159.789,A -85,B 0,C 180,E1 -16576.818,E2 -16576.818} C_VEL
LIN {X 0,Y 291.452,Z 159.793,A -85,B 0,C 180,E1 -16579.875,E2 -16579.875} C_VEL
LIN {X 0,Y 291.384,Z 159.813,A -85,B 0,C 180,E1 -16584.207,E2 -16584.207} C_VEL
LIN {X 0,Y 291.422,Z 159.799,A -85,B 0,C 180,E1 -16587.271,E2 -16587.271} C_VEL
LIN {X 0,Y 291.338,Z 159.79,A -85,B 0,C 180,E1 -16590.437,E2 -16590.437} C_VEL
LIN {X 0,Y 291.345,Z 159.758,A -85,B 0,C 180,E1 -16593.698,E2 -16593.698} C_VEL
LIN {X 0,Y 291.373,Z 159.816,A -85,B 0,C 180,E1 -16597.253,E2 -16597.253} C_VEL
LIN {X 0,Y 291.332,Z 159.778,A -85,B 0,C 180,E1 -16600.642,E2 -16600.642} C_VEL
LIN {X 0,Y 291.291,Z 159.81,A -85,B 0,C 180,E1 -16604.402,E2 -16604.402} C_VEL
LIN {X 0,Y 291.346,Z 160.025,A -85,B 0,C 180,E1 -16606.248,E2 -16606.248} C_VEL
LIN {X 0,Y 293.68,Z 167.509,A -85,B 0,C 180,E1 -16608.958,E2 -16608.958} C_VEL
LIN {X 0,Y 301.764,Z 181.567,A -85,B 0,C 180,E1 -16610.745,E2 -16610.745} C_VEL
LIN {X 0,Y 311.24,Z 199.841,A -85,B 0,C 180,E1 -16612.675,E2 -16612.675} C_VEL
LIN {X 0,Y 319.896,Z 219.428,A -85,B 0,C 180,E1 -16614.378,E2 -16614.378} C_VEL
LIN {X 0,Y 319.698,Z 229.719,A -85,B 0,C 180,E1 -16614.63,E2 -16614.63} C_VEL
LIN {X 0,Y 315.685,Z 333.201,A -85,B 0,C 180,E1 -16616.945,E2 -16616.945} C_VEL
LIN {X 0,Y 314.418,Z 348.603,A -85,B 0,C 180,E1 -16617.51,E2 -16617.51} C_VEL
LIN {X 0,Y 312.638,Z 363.493,A -85,B 0,C 180,E1 -16618.3,E2 -16618.3} C_VEL
LIN {X 0,Y 310.592,Z 377.988,A -85,B 0,C 180,E1 -16619.352,E2 -16619.352} C_VEL
LIN {X 0,Y 308.157,Z 391.889,A -85,B 0,C 180,E1 -16620.637,E2 -16620.637} C_VEL
LIN {X 0,Y 305.307,Z 405.584,A -85,B 0,C 180,E1 -16622.216,E2 -16622.216} C_VEL
LIN {X 0,Y 302.51,Z 417.982,A -85,B 0,C 180,E1 -16623.991,E2 -16623.991} C_VEL
LIN {X 0,Y 299.97,Z 428.732,A -85,B 0,C 180,E1 -16625.868,E2 -16625.868} C_VEL
LIN {X 0,Y 297.74,Z 438.024,A -85,B 0,C 180,E1 -16627.81,E2 -16627.81} C_VEL
LIN {X 0,Y 295.324,Z 447.498,A -85,B 0,C 180,E1 -16630.177,E2 -16630.177} C_VEL
LIN {X 0,Y 293.357,Z 455.391,A -85,B 0,C 180,E1 -16632.574,E2 -16632.574} C_VEL
LIN {X 0,Y 291.754,Z 462.76,A -85,B 0,C 180,E1 -16635.349,E2 -16635.349} C_VEL
LIN {X 0,Y 290.55,Z 468.604,A -85,B 0,C 180,E1 -16638.135,E2 -16638.135} C_VEL
LIN {X 0,Y 290.015,Z 472.079,A -85,B 0,C 180,E1 -16640.233,E2 -16640.233} C_VEL
LIN {X 0,Y 289.566,Z 475.589,A -85,B 0,C 180,E1 -16643.03,E2 -16643.03} C_VEL
LIN {X 0,Y 289.373,Z 477.897,A -85,B 0,C 180,E1 -16645.822,E2 -16645.822} C_VEL
LIN {X 0,Y 289.368,Z 479.056,A -85,B 0,C 180,E1 -16648.608,E2 -16648.608} C_VEL
LIN {X 0,Y 289.368,Z 479.053,A -85,B 0,C 180,E1 -16651.392,E2 -16651.392} C_VEL
LIN {X 0,Y 289.374,Z 477.879,A -85,B 0,C 180,E1 -16654.178,E2 -16654.178} C_VEL
LIN {X 0,Y 289.566,Z 475.559,A -85,B 0,C 180,E1 -16656.97,E2 -16656.97} C_VEL
LIN {X 0,Y 290.01,Z 472.043,A -85,B 0,C 180,E1 -16659.767,E2 -16659.767} C_VEL
LIN {X 0,Y 290.828,Z 467.241,A -85,B 0,C 180,E1 -16662.562,E2 -16662.562} C_VEL
LIN {X 0,Y 292.089,Z 461.023,A -85,B 0,C 180,E1 -16665.347,E2 -16665.347} C_VEL
LIN {X 0,Y 293.895,Z 453.215,A -85,B 0,C 180,E1 -16668.112,E2 -16668.112} C_VEL
LIN {X 0,Y 295.91,Z 444.91,A -85,B 0,C 180,E1 -16670.507,E2 -16670.507} C_VEL
LIN {X 0,Y 298.46,Z 434.921,A -85,B 0,C 180,E1 -16672.86,E2 -16672.86} C_VEL
LIN {X 0,Y 300.909,Z 424.671,A -85,B 0,C 180,E1 -16674.86,E2 -16674.86} C_VEL
LIN {X 0,Y 303.75,Z 412.47,A -85,B 0,C 180,E1 -16676.819,E2 -16676.819} C_VEL
LIN {X 0,Y 306.663,Z 398.88,A -85,B 0,C 180,E1 -16678.581,E2 -16678.581} C_VEL
LIN {X 0,Y 309.318,Z 385.25,A -85,B 0,C 180,E1 -16679.991,E2 -16679.991} C_VEL
LIN {X 0,Y 311.475,Z 371.579,A -85,B 0,C 180,E1 -16681.128,E2 -16681.128} C_VEL
LIN {X 0,Y 313.278,Z 357.892,A -85,B 0,C 180,E1 -16682.005,E2 -16682.005} C_VEL
LIN {X 0,Y 314.898,Z 342.542,A -85,B 0,C 180,E1 -16682.719,E2 -16682.719} C_VEL
LIN {X 0,Y 315.898,Z 327.73,A -85,B 0,C 180,E1 -16683.172,E2 -16683.172} C_VEL
LIN {X 0,Y 319.914,Z 220.312,A -85,B 0,C 180,E1 -16685.564,E2 -16685.564} C_VEL
LIN {X 0,Y 319.376,Z 218.363,A -85,B 0,C 180,E1 -16685.686,E2 -16685.686} C_VEL
LIN {X 0,Y 311.33,Z 200.219,A -85,B 0,C 180,E1 -16687.266,E2 -16687.266} C_VEL
LIN {X 0,Y 303.442,Z 184.747,A -85,B 0,C 180,E1 -16688.863,E2 -16688.863} C_VEL
LIN {X 0,Y 295.884,Z 171.423,A -85,B 0,C 180,E1 -16690.463,E2 -16690.463} C_VEL
LIN {X 0,Y 293.635,Z 167.359,A -85,B 0,C 180,E1 -16691.033,E2 -16691.033} C_VEL
LIN {X 0,Y 291.324,Z 159.953,A -85,B 0,C 180,E1 -16693.748,E2 -16693.748} C_VEL
LIN {X 0,Y 291.319,Z 159.802,A -85,B 0,C 180,E1 -16697.508,E2 -16697.508} C_VEL
LIN {X 0,Y 291.364,Z 159.789,A -85,B 0,C 180,E1 -16701.16,E2 -16701.16} C_VEL
LIN {X 0,Y 291.385,Z 159.781,A -85,B 0,C 180,E1 -16704.63,E2 -16704.63} C_VEL
LIN {X 0,Y 291.372,Z 159.756,A -85,B 0,C 180,E1 -16707.951,E2 -16707.951} C_VEL
LIN {X 0,Y 291.383,Z 159.814,A -85,B 0,C 180,E1 -16711.159,E2 -16711.159} C_VEL
LIN {X 0,Y 291.417,Z 159.792,A -85,B 0,C 180,E1 -16714.272,E2 -16714.272} C_VEL
LIN {X 0,Y 291.383,Z 159.808,A -85,B 0,C 180,E1 -16717.3,E2 -16717.3} C_VEL
LIN {X 0,Y 291.459,Z 159.794,A -85,B 0,C 180,E1 -16720.27,E2 -16720.27} C_VEL
LIN {X 0,Y 291.556,Z 159.771,A -85,B 0,C 180,E1 -16724.624,E2 -16724.624} C_VEL
LIN {X 0,Y 291.531,Z 159.783,A -85,B 0,C 180,E1 -16728.881,E2 -16728.881} C_VEL
LIN {X 0,Y 291.654,Z 159.766,A -85,B 0,C 180,E1 -16731.687,E2 -16731.687} C_VEL
LIN {X 0,Y 291.609,Z 159.776,A -85,B 0,C 180,E1 -16734.468,E2 -16734.468} C_VEL
LIN {X 0,Y 291.886,Z 159.745,A -85,B 0,C 180,E1 -16738.62,E2 -16738.62} C_VEL
LIN {X 0,Y 291.883,Z 159.732,A -85,B 0,C 180,E1 -16741.38,E2 -16741.38} C_VEL
LIN {X 0,Y 291.693,Z 159.766,A -85,B 0,C 180,E1 -16746.919,E2 -16746.919} C_VEL
LIN {X 0,Y 291.569,Z 159.775,A -85,B 0,C 180,E1 -16749.714,E2 -16749.714} C_VEL
LIN {X 0,Y 291.516,Z 159.777,A -85,B 0,C 180,E1 -16753.951,E2 -16753.951} C_VEL
LIN {X 0,Y 291.429,Z 159.807,A -85,B 0,C 180,E1 -16756.821,E2 -16756.821} C_VEL
LIN {X 0,Y 291.392,Z 159.792,A -85,B 0,C 180,E1 -16759.842,E2 -16759.842} C_VEL
LIN {X 0,Y 291.327,Z 159.808,A -85,B 0,C 180,E1 -16764.212,E2 -16764.212} C_VEL
LIN {X 0,Y 291.351,Z 159.817,A -85,B 0,C 180,E1 -16767.279,E2 -16767.279} C_VEL
LIN {X 0,Y 291.318,Z 159.774,A -85,B 0,C 180,E1 -16770.439,E2 -16770.439} C_VEL
LIN {X 0,Y 291.344,Z 159.765,A -85,B 0,C 180,E1 -16773.699,E2 -16773.699} C_VEL
LIN {X 0,Y 291.363,Z 159.811,A -85,B 0,C 180,E1 -16777.25,E2 -16777.25} C_VEL
LIN {X 0,Y 291.295,Z 159.786,A -85,B 0,C 180,E1 -16781.589,E2 -16781.589} C_VEL
LIN {X 0,Y 291.281,Z 159.801,A -85,B 0,C 180,E1 -16785.596,E2 -16785.596} C_VEL
LIN {X 0,Y 291.341,Z 159.982,A -85,B 0,C 180,E1 -16787.511,E2 -16787.511} C_VEL
LIN {X 0,Y 292.402,Z 163.535,A -85,B 0,C 180,E1 -16788.833,E2 -16788.833} C_VEL
LIN {X 0,Y 299.073,Z 174.789,A -85,B 0,C 180,E1 -16790.334,E2 -16790.334} C_VEL
LIN {X 0,Y 305.345,Z 185.888,A -85,B 0,C 180,E1 -16791.633,E2 -16791.633} C_VEL
LIN {X 0,Y 312.137,Z 199.328,A -85,B 0,C 180,E1 -16792.997,E2 -16792.997} C_VEL
LIN {X 0,Y 319.768,Z 216.279,A -85,B 0,C 180,E1 -16794.484,E2 -16794.484} C_VEL
LIN {X 0,Y 320.016,Z 217.642,A -85,B 0,C 180,E1 -16794.553,E2 -16794.553} C_VEL
LIN {X 0,Y 315.744,Z 328.805,A -85,B 0,C 180,E1 -16797.047,E2 -16797.047} C_VEL
LIN {X 0,Y 314.413,Z 344.805,A -85,B 0,C 180,E1 -16797.651,E2 -16797.651} C_VEL
LIN {X 0,Y 312.672,Z 359.965,A -85,B 0,C 180,E1 -16798.494,E2 -16798.494} C_VEL
LIN {X 0,Y 310.558,Z 374.846,A -85,B 0,C 180,E1 -16799.613,E2 -16799.613} C_VEL
LIN {X 0,Y 308.288,Z 387.792,A -85,B 0,C 180,E1 -16800.838,E2 -16800.838} C_VEL
LIN {X 0,Y 305.5,Z 401.279,A -85,B 0,C 180,E1 -16802.421,E2 -16802.421} C_VEL
LIN {X 0,Y 302.731,Z 413.52,A -85,B 0,C 180,E1 -16804.196,E2 -16804.196} C_VEL
LIN {X 0,Y 300.076,Z 425.113,A -85,B 0,C 180,E1 -16806.268,E2 -16806.268} C_VEL
LIN {X 0,Y 297.425,Z 435.508,A -85,B 0,C 180,E1 -16808.515,E2 -16808.515} C_VEL
LIN {X 0,Y 295.184,Z 444.503,A -85,B 0,C 180,E1 -16810.891,E2 -16810.891} C_VEL
LIN {X 0,Y 293.076,Z 452.791,A -85,B 0,C 180,E1 -16813.578,E2 -16813.578} C_VEL
LIN {X 0,Y 291.798,Z 458.927,A -85,B 0,C 180,E1 -16816.063,E2 -16816.063} C_VEL
LIN {X 0,Y 290.621,Z 464.404,A -85,B 0,C 180,E1 -16818.845,E2 -16818.845} C_VEL
LIN {X 0,Y 289.896,Z 468.538,A -85,B 0,C 180,E1 -16821.636,E2 -16821.636} C_VEL
LIN {X 0,Y 289.557,Z 471.443,A -85,B 0,C 180,E1 -16824.429,E2 -16824.429} C_VEL
LIN {X 0,Y 289.437,Z 473.189,A -85,B 0,C 180,E1 -16827.216,E2 -16827.216} C_VEL
LIN {X 0,Y 289.372,Z 473.798,A -85,B 0,C 180,E1 -16830,E2 -16830} C_VEL
LIN {X 0,Y 289.436,Z 473.231,A -85,B 0,C 180,E1 -16832.784,E2 -16832.784} C_VEL
LIN {X 0,Y 289.517,Z 471.54,A -85,B 0,C 180,E1 -16835.572,E2 -16835.572} C_VEL
LIN {X 0,Y 289.876,Z 468.687,A -85,B 0,C 180,E1 -16838.365,E2 -16838.365} C_VEL
LIN {X 0,Y 290.576,Z 464.603,A -85,B 0,C 180,E1 -16841.157,E2 -16841.157} C_VEL
LIN {X 0,Y 291.757,Z 459.188,A -85,B 0,C 180,E1 -16843.939,E2 -16843.939} C_VEL
LIN {X 0,Y 293.252,Z 452.291,A -85,B 0,C 180,E1 -16846.714,E2 -16846.714} C_VEL
LIN {X 0,Y 295.399,Z 443.683,A -85,B 0,C 180,E1 -16849.456,E2 -16849.456} C_VEL
LIN {X 0,Y 297.731,Z 434.532,A -85,B 0,C 180,E1 -16851.826,E2 -16851.826} C_VEL
LIN {X 0,Y 299.69,Z 426.834,A -85,B 0,C 180,E1 -16853.495,E2 -16853.495} C_VEL
LIN {X 0,Y 301.763,Z 418.039,A -85,B 0,C 180,E1 -16855.153,E2 -16855.153} C_VEL
LIN {X 0,Y 304.426,Z 406.706,A -85,B 0,C 180,E1 -16856.941,E2 -16856.941} C_VEL
LIN {X 0,Y 307.036,Z 394.389,A -85,B 0,C 180,E1 -16858.544,E2 -16858.544} C_VEL
LIN {X 0,Y 309.571,Z 380.922,A -85,B 0,C 180,E1 -16859.964,E2 -16859.964} C_VEL
LIN {X 0,Y 311.961,Z 365.906,A -85,B 0,C 180,E1 -16861.209,E2 -16861.209} C_VEL
LIN {X 0,Y 313.78,Z 351.287,A -85,B 0,C 180,E1 -16862.137,E2 -16862.137} C_VEL
LIN {X 0,Y 315.281,Z 336.241,A -85,B 0,C 180,E1 -16862.817,E2 -16862.817} C_VEL
LIN {X 0,Y 316.201,Z 320.581,A -85,B 0,C 180,E1 -16863.279,E2 -16863.279} C_VEL
LIN {X 0,Y 320.102,Z 217.959,A -85,B 0,C 180,E1 -16865.549,E2 -16865.549} C_VEL
LIN {X 0,Y 319.73,Z 216.13,A -85,B 0,C 180,E1 -16865.646,E2 -16865.646} C_VEL
LIN {X 0,Y 312.646,Z 200.356,A -85,B 0,C 180,E1 -16867.028,E2 -16867.028} C_VEL
LIN {X 0,Y 306.001,Z 187.129,A -85,B 0,C 180,E1 -16868.361,E2 -16868.361} C_VEL
LIN {X 0,Y 305.39,Z 185.929,A -85,B 0,C 180,E1 -16868.487,E2 -16868.487} C_VEL
LIN {X 0,Y 302.487,Z 181.767,A -85,B 0,C 180,E1 -16869.051,E2 -16869.051} C_VEL
LIN {X 0,Y 296.571,Z 176.328,A -85,B 0,C 180,E1 -16870.155,E2 -16870.155} C_VEL
LIN {X 0,Y 289.402,Z 170.011,A -85,B 0,C 180,E1 -16871.57,E2 -16871.57} C_VEL
LIN {X 0,Y 287.369,Z 167.429,A -85,B 0,C 180,E1 -16872.016,E2 -16872.016} C_VEL
LIN {X 0,Y 285.085,Z 163.388,A -85,B 0,C 180,E1 -16872.647,E2 -16872.647} C_VEL
LIN {X 0,Y 284.254,Z 160.757,A -85,B 0,C 180,E1 -16873.741,E2 -16873.741} C_VEL
LIN {X 0,Y 284.239,Z 160.671,A -85,B 0,C 180,E1 -16878.118,E2 -16878.118} C_VEL
LIN {X 0,Y 284.288,Z 160.674,A -85,B 0,C 180,E1 -16882.287,E2 -16882.287} C_VEL
LIN {X 0,Y 284.308,Z 160.664,A -85,B 0,C 180,E1 -16885.35,E2 -16885.35} C_VEL
LIN {X 0,Y 284.285,Z 160.635,A -85,B 0,C 180,E1 -16888.724,E2 -16888.724} C_VEL
LIN {X 0,Y 284.283,Z 160.697,A -85,B 0,C 180,E1 -16891.984,E2 -16891.984} C_VEL
LIN {X 0,Y 284.294,Z 160.686,A -85,B 0,C 180,E1 -16896.16,E2 -16896.16} C_VEL
LIN {X 0,Y 284.335,Z 160.671,A -85,B 0,C 180,E1 -16899.928,E2 -16899.928} C_VEL
LIN {X 0,Y 284.446,Z 160.662,A -85,B 0,C 180,E1 -16904.494,E2 -16904.494} C_VEL
LIN {X 0,Y 284.484,Z 160.673,A -85,B 0,C 180,E1 -16908.601,E2 -16908.601} C_VEL
LIN {X 0,Y 284.612,Z 160.633,A -85,B 0,C 180,E1 -16911.48,E2 -16911.48} C_VEL
LIN {X 0,Y 284.577,Z 160.661,A -85,B 0,C 180,E1 -16914.331,E2 -16914.331} C_VEL
LIN {X 0,Y 284.848,Z 160.607,A -85,B 0,C 180,E1 -16918.586,E2 -16918.586} C_VEL
LIN {X 0,Y 284.851,Z 160.621,A -85,B 0,C 180,E1 -16921.414,E2 -16921.414} C_VEL
LIN {X 0,Y 284.648,Z 160.651,A -85,B 0,C 180,E1 -16927.091,E2 -16927.091} C_VEL
LIN {X 0,Y 284.516,Z 160.646,A -85,B 0,C 180,E1 -16929.957,E2 -16929.957} C_VEL
LIN {X 0,Y 284.484,Z 160.659,A -85,B 0,C 180,E1 -16934.303,E2 -16934.303} C_VEL
LIN {X 0,Y 284.425,Z 160.673,A -85,B 0,C 180,E1 -16937.248,E2 -16937.248} C_VEL
LIN {X 0,Y 284.378,Z 160.669,A -85,B 0,C 180,E1 -16940.242,E2 -16940.242} C_VEL
LIN {X 0,Y 284.338,Z 160.681,A -85,B 0,C 180,E1 -16944.846,E2 -16944.846} C_VEL
LIN {X 0,Y 284.332,Z 160.691,A -85,B 0,C 180,E1 -16948.01,E2 -16948.01} C_VEL
LIN {X 0,Y 284.296,Z 160.646,A -85,B 0,C 180,E1 -16951.274,E2 -16951.274} C_VEL
LIN {X 0,Y 284.342,Z 160.657,A -85,B 0,C 180,E1 -16955.348,E2 -16955.348} C_VEL
LIN {X 0,Y 284.309,Z 160.678,A -85,B 0,C 180,E1 -16958.169,E2 -16958.169} C_VEL
LIN {X 0,Y 284.269,Z 160.673,A -85,B 0,C 180,E1 -16962.124,E2 -16962.124} C_VEL
LIN {X 0,Y 284.281,Z 160.924,A -85,B 0,C 180,E1 -16965.2,E2 -16965.2} C_VEL
LIN {X 0,Y 286.454,Z 167.556,A -85,B 0,C 180,E1 -16967.701,E2 -16967.701} C_VEL
LIN {X 0,Y 295.416,Z 182.909,A -85,B 0,C 180,E1 -16969.775,E2 -16969.775} C_VEL
LIN {X 0,Y 303.77,Z 198.706,A -85,B 0,C 180,E1 -16971.561,E2 -16971.561} C_VEL
LIN {X 0,Y 310.849,Z 214.022,A -85,B 0,C 180,E1 -16973.023,E2 -16973.023} C_VEL
LIN {X 0,Y 314.154,Z 221.788,A -85,B 0,C 180,E1 -16973.691,E2 -16973.691} C_VEL
LIN {X 0,Y 310.411,Z 318.417,A -85,B 0,C 180,E1 -16975.87,E2 -16975.87} C_VEL
LIN {X 0,Y 309.448,Z 337.8,A -85,B 0,C 180,E1 -16976.386,E2 -16976.386} C_VEL
LIN {X 0,Y 308.046,Z 352.425,A -85,B 0,C 180,E1 -16976.996,E2 -16976.996} C_VEL
LIN {X 0,Y 306.085,Z 366.901,A -85,B 0,C 180,E1 -16977.832,E2 -16977.832} C_VEL
LIN {X 0,Y 303.959,Z 381.019,A -85,B 0,C 180,E1 -16978.938,E2 -16978.938} C_VEL
LIN {X 0,Y 301.4,Z 394.757,A -85,B 0,C 180,E1 -16980.297,E2 -16980.297} C_VEL
LIN {X 0,Y 298.487,Z 407.903,A -85,B 0,C 180,E1 -16981.907,E2 -16981.907} C_VEL
LIN {X 0,Y 295.872,Z 418.93,A -85,B 0,C 180,E1 -16983.552,E2 -16983.552} C_VEL
LIN {X 0,Y 293.061,Z 430.237,A -85,B 0,C 180,E1 -16985.602,E2 -16985.602} C_VEL
LIN {X 0,Y 290.374,Z 440.879,A -85,B 0,C 180,E1 -16987.966,E2 -16987.966} C_VEL
LIN {X 0,Y 287.971,Z 449.88,A -85,B 0,C 180,E1 -16990.393,E2 -16990.393} C_VEL
LIN {X 0,Y 286.035,Z 457.346,A -85,B 0,C 180,E1 -16992.852,E2 -16992.852} C_VEL
LIN {X 0,Y 284.487,Z 464.31,A -85,B 0,C 180,E1 -16995.697,E2 -16995.697} C_VEL
LIN {X 0,Y 283.295,Z 469.784,A -85,B 0,C 180,E1 -16998.553,E2 -16998.553} C_VEL
LIN {X 0,Y 282.673,Z 473.923,A -85,B 0,C 180,E1 -17001.421,E2 -17001.421} C_VEL
LIN {X 0,Y 282.348,Z 477.113,A -85,B 0,C 180,E1 -17004.653,E2 -17004.653} C_VEL
LIN {X 0,Y 282.29,Z 478.552,A -85,B 0,C 180,E1 -17007.146,E2 -17007.146} C_VEL
LIN {X 0,Y 282.292,Z 479.143,A -85,B 0,C 180,E1 -17010,E2 -17010} C_VEL
LIN {X 0,Y 282.291,Z 478.541,A -85,B 0,C 180,E1 -17012.854,E2 -17012.854} C_VEL
LIN {X 0,Y 282.341,Z 476.797,A -85,B 0,C 180,E1 -17015.714,E2 -17015.714} C_VEL
LIN {X 0,Y 282.672,Z 473.888,A -85,B 0,C 180,E1 -17018.579,E2 -17018.579} C_VEL
LIN {X 0,Y 283.29,Z 469.742,A -85,B 0,C 180,E1 -17021.447,E2 -17021.447} C_VEL
LIN {X 0,Y 284.467,Z 464.25,A -85,B 0,C 180,E1 -17024.303,E2 -17024.303} C_VEL
LIN {X 0,Y 286.031,Z 457.263,A -85,B 0,C 180,E1 -17027.149,E2 -17027.149} C_VEL
LIN {X 0,Y 288.259,Z 448.568,A -85,B 0,C 180,E1 -17029.958,E2 -17029.958} C_VEL
LIN {X 0,Y 290.381,Z 440.775,A -85,B 0,C 180,E1 -17032.033,E2 -17032.033} C_VEL
LIN {X 0,Y 293.041,Z 429.939,A -85,B 0,C 180,E1 -17034.438,E2 -17034.438} C_VEL
LIN {X 0,Y 296.135,Z 417.754,A -85,B 0,C 180,E1 -17036.612,E2 -17036.612} C_VEL
LIN {X 0,Y 299.003,Z 405.324,A -85,B 0,C 180,E1 -17038.423,E2 -17038.423} C_VEL
LIN {X 0,Y 301.635,Z 393.097,A -85,B 0,C 180,E1 -17039.87,E2 -17039.87} C_VEL
LIN {X 0,Y 304.3,Z 378.733,A -85,B 0,C 180,E1 -17041.24,E2 -17041.24} C_VEL
LIN {X 0,Y 306.395,Z 364.274,A -85,B 0,C 180,E1 -17042.326,E2 -17042.326} C_VEL
LIN {X 0,Y 308.337,Z 348.859,A -85,B 0,C 180,E1 -17043.164,E2 -17043.164} C_VEL
LIN {X 0,Y 309.696,Z 333.607,A -85,B 0,C 180,E1 -17043.73,E2 -17043.73} C_VEL
LIN {X 0,Y 314.11,Z 222.451,A -85,B 0,C 180,E1 -17046.263,E2 -17046.263} C_VEL
LIN {X 0,Y 313.654,Z 220.631,A -85,B 0,C 180,E1 -17046.375,E2 -17046.375} C_VEL
LIN {X 0,Y 306.012,Z 203.442,A -85,B 0,C 180,E1 -17047.931,E2 -17047.931} C_VEL
LIN {X 0,Y 298.269,Z 188.158,A -85,B 0,C 180,E1 -17049.562,E2 -17049.562} C_VEL
LIN {X 0,Y 290.974,Z 175.319,A -85,B 0,C 180,E1 -17051.166,E2 -17051.166} C_VEL
LIN {X 0,Y 286.369,Z 167.378,A -85,B 0,C 180,E1 -17052.287,E2 -17052.287} C_VEL
LIN {X 0,Y 284.245,Z 160.789,A -85,B 0,C 180,E1 -17054.847,E2 -17054.847} C_VEL
LIN {X 0,Y 284.271,Z 160.667,A -85,B 0,C 180,E1 -17058.124,E2 -17058.124} C_VEL
LIN {X 0,Y 284.335,Z 160.687,A -85,B 0,C 180,E1 -17062.275,E2 -17062.275} C_VEL
LIN {X 0,Y 284.323,Z 160.642,A -85,B 0,C 180,E1 -17065.353,E2 -17065.353} C_VEL
LIN {X 0,Y 284.296,Z 160.647,A -85,B 0,C 180,E1 -17068.726,E2 -17068.726} C_VEL
LIN {X 0,Y 284.398,Z 160.671,A -85,B 0,C 180,E1 -17072.826,E2 -17072.826} C_VEL
LIN {X 0,Y 284.368,Z 160.688,A -85,B 0,C 180,E1 -17076.707,E2 -17076.707} C_VEL
LIN {X 0,Y 284.405,Z 160.683,A -85,B 0,C 180,E1 -17081.262,E2 -17081.262} C_VEL
LIN {X 0,Y 284.493,Z 160.65,A -85,B 0,C 180,E1 -17084.459,E2 -17084.459} C_VEL
LIN {X 0,Y 284.484,Z 160.664,A -85,B 0,C 180,E1 -17088.601,E2 -17088.601} C_VEL
LIN {X 0,Y 284.611,Z 160.64,A -85,B 0,C 180,E1 -17091.48,E2 -17091.48} C_VEL
LIN {X 0,Y 284.578,Z 160.653,A -85,B 0,C 180,E1 -17094.331,E2 -17094.331} C_VEL
LIN {X 0,Y 284.853,Z 160.62,A -85,B 0,C 180,E1 -17098.586,E2 -17098.586} C_VEL
LIN {X 0,Y 284.849,Z 160.607,A -85,B 0,C 180,E1 -17101.414,E2 -17101.414} C_VEL
LIN {X 0,Y 284.648,Z 160.64,A -85,B 0,C 180,E1 -17107.091,E2 -17107.091} C_VEL
LIN {X 0,Y 284.515,Z 160.656,A -85,B 0,C 180,E1 -17109.957,E2 -17109.957} C_VEL
LIN {X 0,Y 284.464,Z 160.653,A -85,B 0,C 180,E1 -17114.304,E2 -17114.304} C_VEL
LIN {X 0,Y 284.333,Z 160.68,A -85,B 0,C 180,E1 -17118.743,E2 -17118.743} C_VEL
LIN {X 0,Y 284.309,Z 160.693,A -85,B 0,C 180,E1 -17123.298,E2 -17123.298} C_VEL
LIN {X 0,Y 284.327,Z 160.691,A -85,B 0,C 180,E1 -17127.146,E2 -17127.146} C_VEL
LIN {X 0,Y 284.296,Z 160.654,A -85,B 0,C 180,E1 -17130.092,E2 -17130.092} C_VEL
LIN {X 0,Y 284.305,Z 160.631,A -85,B 0,C 180,E1 -17132.946,E2 -17132.946} C_VEL
LIN {X 0,Y 284.325,Z 160.695,A -85,B 0,C 180,E1 -17136.387,E2 -17136.387} C_VEL
LIN {X 0,Y 284.255,Z 160.65,A -85,B 0,C 180,E1 -17140.004,E2 -17140.004} C_VEL
LIN {X 0,Y 284.235,Z 160.695,A -85,B 0,C 180,E1 -17144.188,E2 -17144.188} C_VEL
LIN {X 0,Y 284.293,Z 160.898,A -85,B 0,C 180,E1 -17146.506,E2 -17146.506} C_VEL
LIN {X 0,Y 285.199,Z 163.651,A -85,B 0,C 180,E1 -17147.556,E2 -17147.556} C_VEL
LIN {X 0,Y 294.06,Z 178.41,A -85,B 0,C 180,E1 -17149.63,E2 -17149.63} C_VEL
LIN {X 0,Y 300.856,Z 190.668,A -85,B 0,C 180,E1 -17151.095,E2 -17151.095} C_VEL
LIN {X 0,Y 307.372,Z 203.705,A -85,B 0,C 180,E1 -17152.45,E2 -17152.45} C_VEL
LIN {X 0,Y 314.173,Z 218.923,A -85,B 0,C 180,E1 -17153.824,E2 -17153.824} C_VEL
LIN {X 0,Y 310.405,Z 316.141,A -85,B 0,C 180,E1 -17156.016,E2 -17156.016} C_VEL
LIN {X 0,Y 309.438,Z 333.465,A -85,B 0,C 180,E1 -17156.483,E2 -17156.483} C_VEL
LIN {X 0,Y 308.024,Z 348.69,A -85,B 0,C 180,E1 -17157.139,E2 -17157.139} C_VEL
LIN {X 0,Y 306.345,Z 362.293,A -85,B 0,C 180,E1 -17157.959,E2 -17157.959} C_VEL
LIN {X 0,Y 304.198,Z 376.428,A -85,B 0,C 180,E1 -17159.073,E2 -17159.073} C_VEL
LIN {X 0,Y 301.814,Z 389.294,A -85,B 0,C 180,E1 -17160.342,E2 -17160.342} C_VEL
LIN {X 0,Y 299.206,Z 401.35,A -85,B 0,C 180,E1 -17161.789,E2 -17161.789} C_VEL
LIN {X 0,Y 296.339,Z 413.59,A -85,B 0,C 180,E1 -17163.597,E2 -17163.597} C_VEL
LIN {X 0,Y 293.677,Z 424.563,A -85,B 0,C 180,E1 -17165.579,E2 -17165.579} C_VEL
LIN {X 0,Y 291.178,Z 434.123,A -85,B 0,C 180,E1 -17167.657,E2 -17167.657} C_VEL
LIN {X 0,Y 288.745,Z 443.35,A -85,B 0,C 180,E1 -17170.077,E2 -17170.077} C_VEL
LIN {X 0,Y 286.73,Z 451.022,A -85,B 0,C 180,E1 -17172.527,E2 -17172.527} C_VEL
LIN {X 0,Y 285.215,Z 457.387,A -85,B 0,C 180,E1 -17175.005,E2 -17175.005} C_VEL
LIN {X 0,Y 283.827,Z 463.236,A -85,B 0,C 180,E1 -17177.85,E2 -17177.85} C_VEL
LIN {X 0,Y 283.192,Z 466.698,A -85,B 0,C 180,E1 -17179.996,E2 -17179.996} C_VEL
LIN {X 0,Y 282.6,Z 470.206,A -85,B 0,C 180,E1 -17182.857,E2 -17182.857} C_VEL
LIN {X 0,Y 282.359,Z 472.525,A -85,B 0,C 180,E1 -17185.718,E2 -17185.718} C_VEL
LIN {X 0,Y 282.307,Z 473.707,A -85,B 0,C 180,E1 -17188.574,E2 -17188.574} C_VEL
LIN {X 0,Y 282.307,Z 473.72,A -85,B 0,C 180,E1 -17191.427,E2 -17191.427} C_VEL
LIN {X 0,Y 282.351,Z 472.594,A -85,B 0,C 180,E1 -17194.283,E2 -17194.283} C_VEL
LIN {X 0,Y 282.574,Z 470.329,A -85,B 0,C 180,E1 -17197.144,E2 -17197.144} C_VEL
LIN {X 0,Y 283.172,Z 466.869,A -85,B 0,C 180,E1 -17200.005,E2 -17200.005} C_VEL
LIN {X 0,Y 284.097,Z 462.136,A -85,B 0,C 180,E1 -17202.864,E2 -17202.864} C_VEL
LIN {X 0,Y 285.525,Z 456.003,A -85,B 0,C 180,E1 -17205.709,E2 -17205.709} C_VEL
LIN {X 0,Y 287.479,Z 448.283,A -85,B 0,C 180,E1 -17208.531,E2 -17208.531} C_VEL
LIN {X 0,Y 289.667,Z 440.053,A -85,B 0,C 180,E1 -17210.97,E2 -17210.97} C_VEL
LIN {X 0,Y 292.419,Z 430.138,A -85,B 0,C 180,E1 -17213.364,E2 -17213.364} C_VEL
LIN {X 0,Y 294.86,Z 419.979,A -85,B 0,C 180,E1 -17215.406,E2 -17215.406} C_VEL
LIN {X 0,Y 297.555,Z 408.948,A -85,B 0,C 180,E1 -17217.234,E2 -17217.234} C_VEL
LIN {X 0,Y 300.24,Z 397.039,A -85,B 0,C 180,E1 -17218.868,E2 -17218.868} C_VEL
LIN {X 0,Y 302.808,Z 384.148,A -85,B 0,C 180,E1 -17220.319,E2 -17220.319} C_VEL
LIN {X 0,Y 305.384,Z 369.466,A -85,B 0,C 180,E1 -17221.624,E2 -17221.624} C_VEL
LIN {X 0,Y 307.284,Z 355.296,A -85,B 0,C 180,E1 -17222.609,E2 -17222.609} C_VEL
LIN {X 0,Y 308.992,Z 339.995,A -85,B 0,C 180,E1 -17223.377,E2 -17223.377} C_VEL
LIN {X 0,Y 310.081,Z 325.218,A -85,B 0,C 180,E1 -17223.878,E2 -17223.878} C_VEL
LIN {X 0,Y 314.259,Z 219.705,A -85,B 0,C 180,E1 -17226.267,E2 -17226.267} C_VEL
LIN {X 0,Y 313.625,Z 217.573,A -85,B 0,C 180,E1 -17226.411,E2 -17226.411} C_VEL
LIN {X 0,Y 306.38,Z 201.495,A -85,B 0,C 180,E1 -17227.885,E2 -17227.885} C_VEL
LIN {X 0,Y 298.009,Z 185.255,A -85,B 0,C 180,E1 -17229.647,E2 -17229.647} C_VEL
LIN {X 0,Y 290.124,Z 171.886,A -85,B 0,C 180,E1 -17231.383,E2 -17231.383} C_VEL
LIN {X 0,Y 287.369,Z 167.429,A -85,B 0,C 180,E1 -17232.016,E2 -17232.016} C_VEL
LIN {X 0,Y 285.136,Z 165.142,A -85,B 0,C 180,E1 -17232.515,E2 -17232.515} C_VEL
LIN {X 0,Y 282.63,Z 163.705,A -85,B 0,C 180,E1 -17233.105,E2 -17233.105} C_VEL
LIN {X 0,Y 278.904,Z 162.204,A -85,B 0,C 180,E1 -17234.254,E2 -17234.254} C_VEL
LIN {X 0,Y 277.352,Z 161.63,A -85,B 0,C 180,E1 -17235.184,E2 -17235.184} C_VEL
LIN {X 0,Y 277.16,Z 161.567,A -85,B 0,C 180,E1 -17235.606,E2 -17235.606} C_VEL
LIN {X 0,Y 277.177,Z 161.532,A -85,B 0,C 180,E1 -17239.523,E2 -17239.523} C_VEL
LIN {X 0,Y 277.239,Z 161.556,A -85,B 0,C 180,E1 -17242.526,E2 -17242.526} C_VEL
LIN {X 0,Y 277.247,Z 161.524,A -85,B 0,C 180,E1 -17246.104,E2 -17246.104} C_VEL
LIN {X 0,Y 277.246,Z 161.52,A -85,B 0,C 180,E1 -17249.536,E2 -17249.536} C_VEL
LIN {X 0,Y 277.29,Z 161.569,A -85,B 0,C 180,E1 -17252.857,E2 -17252.857} C_VEL
LIN {X 0,Y 277.257,Z 161.561,A -85,B 0,C 180,E1 -17256.073,E2 -17256.073} C_VEL
LIN {X 0,Y 277.284,Z 161.551,A -85,B 0,C 180,E1 -17260.762,E2 -17260.762} C_VEL
LIN {X 0,Y 277.41,Z 161.532,A -85,B 0,C 180,E1 -17265.324,E2 -17265.324} C_VEL
LIN {X 0,Y 277.459,Z 161.539,A -85,B 0,C 180,E1 -17269.787,E2 -17269.787} C_VEL
LIN {X 0,Y 277.606,Z 161.513,A -85,B 0,C 180,E1 -17272.728,E2 -17272.728} C_VEL
LIN {X 0,Y 277.814,Z 161.482,A -85,B 0,C 180,E1 -17278.55,E2 -17278.55} C_VEL
LIN {X 0,Y 277.817,Z 161.496,A -85,B 0,C 180,E1 -17281.449,E2 -17281.449} C_VEL
LIN {X 0,Y 277.606,Z 161.526,A -85,B 0,C 180,E1 -17287.272,E2 -17287.272} C_VEL
LIN {X 0,Y 277.459,Z 161.525,A -85,B 0,C 180,E1 -17290.213,E2 -17290.213} C_VEL
LIN {X 0,Y 277.436,Z 161.532,A -85,B 0,C 180,E1 -17294.674,E2 -17294.674} C_VEL
LIN {X 0,Y 277.344,Z 161.557,A -85,B 0,C 180,E1 -17299.234,E2 -17299.234} C_VEL
LIN {X 0,Y 277.293,Z 161.567,A -85,B 0,C 180,E1 -17304.157,E2 -17304.157} C_VEL
LIN {X 0,Y 277.326,Z 161.557,A -85,B 0,C 180,E1 -17307.504,E2 -17307.504} C_VEL
LIN {X 0,Y 277.273,Z 161.536,A -85,B 0,C 180,E1 -17310.481,E2 -17310.481} C_VEL
LIN {X 0,Y 277.247,Z 161.513,A -85,B 0,C 180,E1 -17313.895,E2 -17313.895} C_VEL
LIN {X 0,Y 277.266,Z 161.57,A -85,B 0,C 180,E1 -17317.469,E2 -17317.469} C_VEL
LIN {X 0,Y 277.209,Z 161.539,A -85,B 0,C 180,E1 -17321.236,E2 -17321.236} C_VEL
LIN {X 0,Y 277.228,Z 161.742,A -85,B 0,C 180,E1 -17324.047,E2 -17324.047} C_VEL
LIN {X 0,Y 279.108,Z 167.465,A -85,B 0,C 180,E1 -17326.314,E2 -17326.314} C_VEL
LIN {X 0,Y 286.085,Z 179.101,A -85,B 0,C 180,E1 -17328.052,E2 -17328.052} C_VEL
LIN {X 0,Y 292.663,Z 190.581,A -85,B 0,C 180,E1 -17329.561,E2 -17329.561} C_VEL
LIN {X 0,Y 301.406,Z 207.842,A -85,B 0,C 180,E1 -17331.477,E2 -17331.477} C_VEL
LIN {X 0,Y 308.426,Z 223.995,A -85,B 0,C 180,E1 -17332.969,E2 -17332.969} C_VEL
LIN {X 0,Y 303.904,Z 333.102,A -85,B 0,C 180,E1 -17335.488,E2 -17335.488} C_VEL
LIN {X 0,Y 302.539,Z 348.491,A -85,B 0,C 180,E1 -17336.065,E2 -17336.065} C_VEL
LIN {X 0,Y 300.638,Z 363.376,A -85,B 0,C 180,E1 -17336.877,E2 -17336.877} C_VEL
LIN {X 0,Y 298.362,Z 378.3,A -85,B 0,C 180,E1 -17337.993,E2 -17337.993} C_VEL
LIN {X 0,Y 295.807,Z 391.765,A -85,B 0,C 180,E1 -17339.282,E2 -17339.282} C_VEL
LIN {X 0,Y 292.786,Z 405.459,A -85,B 0,C 180,E1 -17340.917,E2 -17340.917} C_VEL
LIN {X 0,Y 289.781,Z 417.855,A -85,B 0,C 180,E1 -17342.756,E2 -17342.756} C_VEL
LIN {X 0,Y 287.074,Z 428.247,A -85,B 0,C 180,E1 -17344.632,E2 -17344.632} C_VEL
LIN {X 0,Y 284.552,Z 437.894,A -85,B 0,C 180,E1 -17346.723,E2 -17346.723} C_VEL
LIN {X 0,Y 281.893,Z 447.368,A -85,B 0,C 180,E1 -17349.19,E2 -17349.19} C_VEL
LIN {X 0,Y 279.741,Z 455.26,A -85,B 0,C 180,E1 -17351.697,E2 -17351.697} C_VEL
LIN {X 0,Y 277.933,Z 462.629,A -85,B 0,C 180,E1 -17354.603,E2 -17354.603} C_VEL
LIN {X 0,Y 276.581,Z 468.472,A -85,B 0,C 180,E1 -17357.526,E2 -17357.526} C_VEL
LIN {X 0,Y 275.915,Z 471.947,A -85,B 0,C 180,E1 -17359.729,E2 -17359.729} C_VEL
LIN {X 0,Y 275.414,Z 475.457,A -85,B 0,C 180,E1 -17362.67,E2 -17362.67} C_VEL
LIN {X 0,Y 275.2,Z 477.765,A -85,B 0,C 180,E1 -17365.606,E2 -17365.606} C_VEL
LIN {X 0,Y 275.218,Z 478.924,A -85,B 0,C 180,E1 -17368.537,E2 -17368.537} C_VEL
LIN {X 0,Y 275.218,Z 478.921,A -85,B 0,C 180,E1 -17371.463,E2 -17371.463} C_VEL
LIN {X 0,Y 275.2,Z 477.745,A -85,B 0,C 180,E1 -17374.394,E2 -17374.394} C_VEL
LIN {X 0,Y 275.414,Z 475.425,A -85,B 0,C 180,E1 -17377.33,E2 -17377.33} C_VEL
LIN {X 0,Y 275.911,Z 471.907,A -85,B 0,C 180,E1 -17380.271,E2 -17380.271} C_VEL
LIN {X 0,Y 276.885,Z 467.105,A -85,B 0,C 180,E1 -17383.205,E2 -17383.205} C_VEL
LIN {X 0,Y 278.255,Z 460.886,A -85,B 0,C 180,E1 -17386.131,E2 -17386.131} C_VEL
LIN {X 0,Y 280.314,Z 453.078,A -85,B 0,C 180,E1 -17389.022,E2 -17389.022} C_VEL
LIN {X 0,Y 282.535,Z 444.772,A -85,B 0,C 180,E1 -17391.525,E2 -17391.525} C_VEL
LIN {X 0,Y 285.132,Z 435.447,A -85,B 0,C 180,E1 -17393.829,E2 -17393.829} C_VEL
LIN {X 0,Y 288,Z 424.532,A -85,B 0,C 180,E1 -17396.056,E2 -17396.056} C_VEL
LIN {X 0,Y 291.091,Z 412.331,A -85,B 0,C 180,E1 -17398.086,E2 -17398.086} C_VEL
LIN {X 0,Y 293.939,Z 400.081,A -85,B 0,C 180,E1 -17399.744,E2 -17399.744} C_VEL
LIN {X 0,Y 296.751,Z 386.744,A -85,B 0,C 180,E1 -17401.203,E2 -17401.203} C_VEL
LIN {X 0,Y 299.079,Z 373.35,A -85,B 0,C 180,E1 -17402.382,E2 -17402.382} C_VEL
LIN {X 0,Y 301.132,Z 359.043,A -85,B 0,C 180,E1 -17403.361,E2 -17403.361} C_VEL
LIN {X 0,Y 302.866,Z 344.22,A -85,B 0,C 180,E1 -17404.093,E2 -17404.093} C_VEL
LIN {X 0,Y 304.007,Z 329.068,A -85,B 0,C 180,E1 -17404.599,E2 -17404.599} C_VEL
LIN {X 0,Y 308.342,Z 223.872,A -85,B 0,C 180,E1 -17407.01,E2 -17407.01} C_VEL
LIN {X 0,Y 300.579,Z 206.337,A -85,B 0,C 180,E1 -17408.654,E2 -17408.654} C_VEL
LIN {X 0,Y 293.264,Z 191.837,A -85,B 0,C 180,E1 -17410.256,E2 -17410.256} C_VEL
LIN {X 0,Y 286.748,Z 180.206,A -85,B 0,C 180,E1 -17411.745,E2 -17411.745} C_VEL
LIN {X 0,Y 281.153,Z 170.997,A -85,B 0,C 180,E1 -17413.082,E2 -17413.082} C_VEL
LIN {X 0,Y 278.961,Z 167.124,A -85,B 0,C 180,E1 -17413.719,E2 -17413.719} C_VEL
LIN {X 0,Y 277.224,Z 161.656,A -85,B 0,C 180,E1 -17415.965,E2 -17415.965} C_VEL
LIN {X 0,Y 277.222,Z 161.533,A -85,B 0,C 180,E1 -17419.512,E2 -17419.512} C_VEL
LIN {X 0,Y 277.282,Z 161.57,A -85,B 0,C 180,E1 -17422.533,E2 -17422.533} C_VEL
LIN {X 0,Y 277.254,Z 161.511,A -85,B 0,C 180,E1 -17426.105,E2 -17426.105} C_VEL
LIN {X 0,Y 277.262,Z 161.54,A -85,B 0,C 180,E1 -17429.539,E2 -17429.539} C_VEL
LIN {X 0,Y 277.36,Z 161.547,A -85,B 0,C 180,E1 -17432.864,E2 -17432.864} C_VEL
LIN {X 0,Y 277.339,Z 161.563,A -85,B 0,C 180,E1 -17436.081,E2 -17436.081} C_VEL
LIN {X 0,Y 277.346,Z 161.557,A -85,B 0,C 180,E1 -17440.766,E2 -17440.766} C_VEL
LIN {X 0,Y 277.436,Z 161.532,A -85,B 0,C 180,E1 -17445.326,E2 -17445.326} C_VEL
LIN {X 0,Y 277.458,Z 161.525,A -85,B 0,C 180,E1 -17449.787,E2 -17449.787} C_VEL
LIN {X 0,Y 277.605,Z 161.526,A -85,B 0,C 180,E1 -17452.728,E2 -17452.728} C_VEL
LIN {X 0,Y 277.819,Z 161.496,A -85,B 0,C 180,E1 -17458.551,E2 -17458.551} C_VEL
LIN {X 0,Y 277.815,Z 161.482,A -85,B 0,C 180,E1 -17461.45,E2 -17461.45} C_VEL
LIN {X 0,Y 277.606,Z 161.514,A -85,B 0,C 180,E1 -17467.272,E2 -17467.272} C_VEL
LIN {X 0,Y 277.459,Z 161.538,A -85,B 0,C 180,E1 -17470.213,E2 -17470.213} C_VEL
LIN {X 0,Y 277.41,Z 161.531,A -85,B 0,C 180,E1 -17474.676,E2 -17474.676} C_VEL
LIN {X 0,Y 277.285,Z 161.552,A -85,B 0,C 180,E1 -17479.238,E2 -17479.238} C_VEL
LIN {X 0,Y 277.256,Z 161.563,A -85,B 0,C 180,E1 -17483.927,E2 -17483.927} C_VEL
LIN {X 0,Y 277.268,Z 161.573,A -85,B 0,C 180,E1 -17487.482,E2 -17487.482} C_VEL
LIN {X 0,Y 277.249,Z 161.522,A -85,B 0,C 180,E1 -17490.473,E2 -17490.473} C_VEL
LIN {X 0,Y 277.246,Z 161.521,A -85,B 0,C 180,E1 -17493.896,E2 -17493.896} C_VEL
LIN {X 0,Y 277.239,Z 161.56,A -85,B 0,C 180,E1 -17497.474,E2 -17497.474} C_VEL
LIN {X 0,Y 277.177,Z 161.537,A -85,B 0,C 180,E1 -17501.243,E2 -17501.243} C_VEL
LIN {X 0,Y 277.214,Z 161.743,A -85,B 0,C 180,E1 -17505.364,E2 -17505.364} C_VEL
LIN {X 0,Y 277.811,Z 163.676,A -85,B 0,C 180,E1 -17506.131,E2 -17506.131} C_VEL
LIN {X 0,Y 284.338,Z 174.12,A -85,B 0,C 180,E1 -17507.795,E2 -17507.795} C_VEL
LIN {X 0,Y 292.892,Z 188.749,A -85,B 0,C 180,E1 -17509.762,E2 -17509.762} C_VEL
LIN {X 0,Y 301.008,Z 204.612,A -85,B 0,C 180,E1 -17511.536,E2 -17511.536} C_VEL
LIN {X 0,Y 307.666,Z 219.349,A -85,B 0,C 180,E1 -17512.942,E2 -17512.942} C_VEL
LIN {X 0,Y 308.376,Z 221.075,A -85,B 0,C 180,E1 -17513.091,E2 -17513.091} C_VEL
LIN {X 0,Y 304.558,Z 316.231,A -85,B 0,C 180,E1 -17515.271,E2 -17515.271} C_VEL
LIN {X 0,Y 303.568,Z 333.546,A -85,B 0,C 180,E1 -17515.746,E2 -17515.746} C_VEL
LIN {X 0,Y 302.082,Z 348.766,A -85,B 0,C 180,E1 -17516.408,E2 -17516.408} C_VEL
LIN {X 0,Y 300.331,Z 362.367,A -85,B 0,C 180,E1 -17517.238,E2 -17517.238} C_VEL
LIN {X 0,Y 298.076,Z 376.787,A -85,B 0,C 180,E1 -17518.398,E2 -17518.398} C_VEL
LIN {X 0,Y 295.353,Z 390.79,A -85,B 0,C 180,E1 -17519.823,E2 -17519.823} C_VEL
LIN {X 0,Y 292.4,Z 403.763,A -85,B 0,C 180,E1 -17521.464,E2 -17521.464} C_VEL
LIN {X 0,Y 289.444,Z 415.609,A -85,B 0,C 180,E1 -17523.308,E2 -17523.308} C_VEL
LIN {X 0,Y 286.739,Z 426.449,A -85,B 0,C 180,E1 -17525.375,E2 -17525.375} C_VEL
LIN {X 0,Y 284.196,Z 435.646,A -85,B 0,C 180,E1 -17527.461,E2 -17527.461} C_VEL
LIN {X 0,Y 281.709,Z 444.64,A -85,B 0,C 180,E1 -17529.938,E2 -17529.938} C_VEL
LIN {X 0,Y 279.642,Z 452.095,A -85,B 0,C 180,E1 -17532.447,E2 -17532.447} C_VEL
LIN {X 0,Y 277.949,Z 459.063,A -85,B 0,C 180,E1 -17535.354,E2 -17535.354} C_VEL
LIN {X 0,Y 276.595,Z 464.54,A -85,B 0,C 180,E1 -17538.272,E2 -17538.272} C_VEL
LIN {X 0,Y 275.811,Z 468.673,A -85,B 0,C 180,E1 -17541.206,E2 -17541.206} C_VEL
LIN {X 0,Y 275.359,Z 471.854,A -85,B 0,C 180,E1 -17544.504,E2 -17544.504} C_VEL
LIN {X 0,Y 275.257,Z 473.322,A -85,B 0,C 180,E1 -17547.073,E2 -17547.073} C_VEL
LIN {X 0,Y 275.22,Z 473.931,A -85,B 0,C 180,E1 -17550,E2 -17550} C_VEL
LIN {X 0,Y 275.255,Z 473.363,A -85,B 0,C 180,E1 -17552.927,E2 -17552.927} C_VEL
LIN {X 0,Y 275.377,Z 471.672,A -85,B 0,C 180,E1 -17555.859,E2 -17555.859} C_VEL
LIN {X 0,Y 275.796,Z 468.818,A -85,B 0,C 180,E1 -17558.795,E2 -17558.795} C_VEL
LIN {X 0,Y 276.564,Z 464.734,A -85,B 0,C 180,E1 -17561.73,E2 -17561.73} C_VEL
LIN {X 0,Y 277.911,Z 459.319,A -85,B 0,C 180,E1 -17564.649,E2 -17564.649} C_VEL
LIN {X 0,Y 279.607,Z 452.421,A -85,B 0,C 180,E1 -17567.555,E2 -17567.555} C_VEL
LIN {X 0,Y 281.954,Z 443.812,A -85,B 0,C 180,E1 -17570.424,E2 -17570.424} C_VEL
LIN {X 0,Y 284.57,Z 434.66,A -85,B 0,C 180,E1 -17572.891,E2 -17572.891} C_VEL
LIN {X 0,Y 287.114,Z 424.882,A -85,B 0,C 180,E1 -17575.083,E2 -17575.083} C_VEL
LIN {X 0,Y 290.172,Z 413.277,A -85,B 0,C 180,E1 -17577.204,E2 -17577.204} C_VEL
LIN {X 0,Y 293.125,Z 400.96,A -85,B 0,C 180,E1 -17579.046,E2 -17579.046} C_VEL
LIN {X 0,Y 296.112,Z 387.367,A -85,B 0,C 180,E1 -17580.683,E2 -17580.683} C_VEL
LIN {X 0,Y 298.519,Z 374.643,A -85,B 0,C 180,E1 -17581.915,E2 -17581.915} C_VEL
LIN {X 0,Y 300.639,Z 360.38,A -85,B 0,C 180,E1 -17583.023,E2 -17583.023} C_VEL
LIN {X 0,Y 302.56,Z 345.31,A -85,B 0,C 180,E1 -17583.882,E2 -17583.882} C_VEL
LIN {X 0,Y 303.948,Z 329.528,A -85,B 0,C 180,E1 -17584.507,E2 -17584.507} C_VEL
LIN {X 0,Y 307.074,Z 256.641,A -85,B 0,C 180,E1 -17586.202,E2 -17586.202} C_VEL
LIN {X 0,Y 308.399,Z 220.967,A -85,B 0,C 180,E1 -17587.035,E2 -17587.035} C_VEL
LIN {X 0,Y 301.229,Z 204.944,A -85,B 0,C 180,E1 -17588.55,E2 -17588.55} C_VEL
LIN {X 0,Y 293.198,Z 189.311,A -85,B 0,C 180,E1 -17590.304,E2 -17590.304} C_VEL
LIN {X 0,Y 285.5,Z 176.103,A -85,B 0,C 180,E1 -17592.066,E2 -17592.066} C_VEL
LIN {X 0,Y 279.931,Z 167.255,A -85,B 0,C 180,E1 -17593.411,E2 -17593.411} C_VEL
LIN {X 0,Y 277.725,Z 163.462,A -85,B 0,C 180,E1 -17594.069,E2 -17594.069} C_VEL
LIN {X 0,Y 277.176,Z 161.623,A -85,B 0,C 180,E1 -17594.915,E2 -17594.915} C_VEL
LIN {X 0,Y 277.16,Z 161.567,A -85,B 0,C 180,E1 -17595.606,E2 -17595.606} C_VEL
LIN {X 0,Y 276.481,Z 161.67,A -85,B 0,C 180,E1 -17596.818,E2 -17596.818} C_VEL
LIN {X 0,Y 273.636,Z 161.991,A -85,B 0,C 180,E1 -17598.795,E2 -17598.795} C_VEL
LIN {X 0,Y 271.236,Z 162.277,A -85,B 0,C 180,E1 -17600.4,E2 -17600.4} C_VEL
LIN {X 0,Y 270.216,Z 162.41,A -85,B 0,C 180,E1 -17601.645,E2 -17601.645} C_VEL
LIN {X 0,Y 270.138,Z 162.427,A -85,B 0,C 180,E1 -17602.066,E2 -17602.066} C_VEL
LIN {X 0,Y 270.2,Z 162.424,A -85,B 0,C 180,E1 -17605.094,E2 -17605.094} C_VEL
LIN {X 0,Y 270.185,Z 162.392,A -85,B 0,C 180,E1 -17609.136,E2 -17609.136} C_VEL
LIN {X 0,Y 270.223,Z 162.45,A -85,B 0,C 180,E1 -17612.163,E2 -17612.163} C_VEL
LIN {X 0,Y 270.185,Z 162.454,A -85,B 0,C 180,E1 -17617.034,E2 -17617.034} C_VEL
LIN {X 0,Y 270.224,Z 162.428,A -85,B 0,C 180,E1 -17620.238,E2 -17620.238} C_VEL
LIN {X 0,Y 270.369,Z 162.41,A -85,B 0,C 180,E1 -17624.933,E2 -17624.933} C_VEL
LIN {X 0,Y 270.411,Z 162.419,A -85,B 0,C 180,E1 -17629.518,E2 -17629.518} C_VEL
LIN {X 0,Y 270.567,Z 162.387,A -85,B 0,C 180,E1 -17632.537,E2 -17632.537} C_VEL
LIN {X 0,Y 270.779,Z 162.357,A -85,B 0,C 180,E1 -17638.513,E2 -17638.513} C_VEL
LIN {X 0,Y 270.783,Z 162.372,A -85,B 0,C 180,E1 -17641.487,E2 -17641.487} C_VEL
LIN {X 0,Y 270.567,Z 162.401,A -85,B 0,C 180,E1 -17647.462,E2 -17647.462} C_VEL
LIN {X 0,Y 270.412,Z 162.404,A -85,B 0,C 180,E1 -17650.482,E2 -17650.482} C_VEL
LIN {X 0,Y 270.405,Z 162.405,A -85,B 0,C 180,E1 -17655.064,E2 -17655.064} C_VEL
LIN {X 0,Y 270.302,Z 162.427,A -85,B 0,C 180,E1 -17659.755,E2 -17659.755} C_VEL
LIN {X 0,Y 270.239,Z 162.439,A -85,B 0,C 180,E1 -17664.589,E2 -17664.589} C_VEL
LIN {X 0,Y 270.273,Z 162.441,A -85,B 0,C 180,E1 -17667.908,E2 -17667.908} C_VEL
LIN {X 0,Y 270.185,Z 162.399,A -85,B 0,C 180,E1 -17671.348,E2 -17671.348} C_VEL
LIN {X 0,Y 270.202,Z 162.404,A -85,B 0,C 180,E1 -17674.905,E2 -17674.905} C_VEL
LIN {X 0,Y 270.198,Z 162.422,A -85,B 0,C 180,E1 -17678.71,E2 -17678.71} C_VEL
LIN {X 0,Y 270.192,Z 162.618,A -85,B 0,C 180,E1 -17682.838,E2 -17682.838} C_VEL
LIN {X 0,Y 271.672,Z 167.206,A -85,B 0,C 180,E1 -17684.771,E2 -17684.771} C_VEL
LIN {X 0,Y 274.648,Z 172,A -85,B 0,C 180,E1 -17685.619,E2 -17685.619} C_VEL
LIN {X 0,Y 281.406,Z 183.039,A -85,B 0,C 180,E1 -17687.325,E2 -17687.325} C_VEL
LIN {X 0,Y 288.827,Z 196.425,A -85,B 0,C 180,E1 -17689.099,E2 -17689.099} C_VEL
LIN {X 0,Y 296.817,Z 212.535,A -85,B 0,C 180,E1 -17690.913,E2 -17690.913} C_VEL
LIN {X 0,Y 302.681,Z 226.136,A -85,B 0,C 180,E1 -17692.208,E2 -17692.208} C_VEL
LIN {X 0,Y 298.237,Z 330.052,A -85,B 0,C 180,E1 -17694.632,E2 -17694.632} C_VEL
LIN {X 0,Y 296.99,Z 345.693,A -85,B 0,C 180,E1 -17695.187,E2 -17695.187} C_VEL
LIN {X 0,Y 295.09,Z 360.715,A -85,B 0,C 180,E1 -17695.966,E2 -17695.966} C_VEL
LIN {X 0,Y 293.111,Z 373.54,A -85,B 0,C 180,E1 -17696.866,E2 -17696.866} C_VEL
LIN {X 0,Y 290.681,Z 386.956,A -85,B 0,C 180,E1 -17698.069,E2 -17698.069} C_VEL
LIN {X 0,Y 287.838,Z 400.23,A -85,B 0,C 180,E1 -17699.559,E2 -17699.559} C_VEL
LIN {X 0,Y 284.803,Z 412.438,A -85,B 0,C 180,E1 -17701.236,E2 -17701.236} C_VEL
LIN {X 0,Y 281.592,Z 424.613,A -85,B 0,C 180,E1 -17703.305,E2 -17703.305} C_VEL
LIN {X 0,Y 278.551,Z 435.643,A -85,B 0,C 180,E1 -17705.609,E2 -17705.609} C_VEL
LIN {X 0,Y 275.885,Z 444.816,A -85,B 0,C 180,E1 -17707.929,E2 -17707.929} C_VEL
LIN {X 0,Y 273.558,Z 453.107,A -85,B 0,C 180,E1 -17710.489,E2 -17710.489} C_VEL
LIN {X 0,Y 271.407,Z 460.895,A -85,B 0,C 180,E1 -17713.451,E2 -17713.451} C_VEL
LIN {X 0,Y 269.928,Z 467.091,A -85,B 0,C 180,E1 -17716.448,E2 -17716.448} C_VEL
LIN {X 0,Y 268.882,Z 471.881,A -85,B 0,C 180,E1 -17719.457,E2 -17719.457} C_VEL
LIN {X 0,Y 268.333,Z 475.391,A -85,B 0,C 180,E1 -17722.475,E2 -17722.475} C_VEL
LIN {X 0,Y 268.102,Z 477.698,A -85,B 0,C 180,E1 -17725.489,E2 -17725.489} C_VEL
LIN {X 0,Y 268.124,Z 478.858,A -85,B 0,C 180,E1 -17728.498,E2 -17728.498} C_VEL
LIN {X 0,Y 268.124,Z 478.854,A -85,B 0,C 180,E1 -17731.502,E2 -17731.502} C_VEL
LIN {X 0,Y 268.102,Z 477.679,A -85,B 0,C 180,E1 -17734.51,E2 -17734.51} C_VEL
LIN {X 0,Y 268.333,Z 475.357,A -85,B 0,C 180,E1 -17737.525,E2 -17737.525} C_VEL
LIN {X 0,Y 268.877,Z 471.84,A -85,B 0,C 180,E1 -17740.543,E2 -17740.543} C_VEL
LIN {X 0,Y 269.92,Z 467.037,A -85,B 0,C 180,E1 -17743.552,E2 -17743.552} C_VEL
LIN {X 0,Y 271.431,Z 460.551,A -85,B 0,C 180,E1 -17746.661,E2 -17746.661} C_VEL
LIN {X 0,Y 273.552,Z 453.009,A -85,B 0,C 180,E1 -17749.511,E2 -17749.511} C_VEL
LIN {X 0,Y 275.887,Z 444.703,A -85,B 0,C 180,E1 -17752.07,E2 -17752.07} C_VEL
LIN {X 0,Y 278.512,Z 435.637,A -85,B 0,C 180,E1 -17754.363,E2 -17754.363} C_VEL
LIN {X 0,Y 281.079,Z 426.246,A -85,B 0,C 180,E1 -17756.347,E2 -17756.347} C_VEL
LIN {X 0,Y 284.242,Z 414.404,A -85,B 0,C 180,E1 -17758.422,E2 -17758.422} C_VEL
LIN {X 0,Y 287.144,Z 402.597,A -85,B 0,C 180,E1 -17760.116,E2 -17760.116} C_VEL
LIN {X 0,Y 290.047,Z 389.841,A -85,B 0,C 180,E1 -17761.6,E2 -17761.6} C_VEL
LIN {X 0,Y 292.443,Z 377.099,A -85,B 0,C 180,E1 -17762.815,E2 -17762.815} C_VEL
LIN {X 0,Y 294.702,Z 362.87,A -85,B 0,C 180,E1 -17763.879,E2 -17763.879} C_VEL
LIN {X 0,Y 296.635,Z 347.809,A -85,B 0,C 180,E1 -17764.705,E2 -17764.705} C_VEL
LIN {X 0,Y 298.055,Z 331.997,A -85,B 0,C 180,E1 -17765.289,E2 -17765.289} C_VEL
LIN {X 0,Y 302.598,Z 225.941,A -85,B 0,C 180,E1 -17767.771,E2 -17767.771} C_VEL
LIN {X 0,Y 294.543,Z 207.777,A -85,B 0,C 180,E1 -17769.551,E2 -17769.551} C_VEL
LIN {X 0,Y 285.752,Z 190.659,A -85,B 0,C 180,E1 -17771.578,E2 -17771.578} C_VEL
LIN {X 0,Y 277.386,Z 176.428,A -85,B 0,C 180,E1 -17773.621,E2 -17773.621} C_VEL
LIN {X 0,Y 273.875,Z 171.027,A -85,B 0,C 180,E1 -17774.517,E2 -17774.517} C_VEL
LIN {X 0,Y 271.588,Z 167.036,A -85,B 0,C 180,E1 -17775.221,E2 -17775.221} C_VEL
LIN {X 0,Y 270.195,Z 162.537,A -85,B 0,C 180,E1 -17777.162,E2 -17777.162} C_VEL
LIN {X 0,Y 270.207,Z 162.424,A -85,B 0,C 180,E1 -17781.374,E2 -17781.374} C_VEL
LIN {X 0,Y 270.215,Z 162.401,A -85,B 0,C 180,E1 -17785.097,E2 -17785.097} C_VEL
LIN {X 0,Y 270.201,Z 162.407,A -85,B 0,C 180,E1 -17789.131,E2 -17789.131} C_VEL
LIN {X 0,Y 270.266,Z 162.44,A -85,B 0,C 180,E1 -17792.146,E2 -17792.146} C_VEL
LIN {X 0,Y 270.281,Z 162.436,A -85,B 0,C 180,E1 -17795.518,E2 -17795.518} C_VEL
LIN {X 0,Y 270.303,Z 162.427,A -85,B 0,C 180,E1 -17800.245,E2 -17800.245} C_VEL
LIN {X 0,Y 270.404,Z 162.405,A -85,B 0,C 180,E1 -17804.936,E2 -17804.936} C_VEL
LIN {X 0,Y 270.411,Z 162.404,A -85,B 0,C 180,E1 -17809.518,E2 -17809.518} C_VEL
LIN {X 0,Y 270.566,Z 162.401,A -85,B 0,C 180,E1 -17812.538,E2 -17812.538} C_VEL
LIN {X 0,Y 270.785,Z 162.371,A -85,B 0,C 180,E1 -17818.513,E2 -17818.513} C_VEL
LIN {X 0,Y 270.779,Z 162.357,A -85,B 0,C 180,E1 -17821.487,E2 -17821.487} C_VEL
LIN {X 0,Y 270.567,Z 162.387,A -85,B 0,C 180,E1 -17827.463,E2 -17827.463} C_VEL
LIN {X 0,Y 270.411,Z 162.418,A -85,B 0,C 180,E1 -17830.482,E2 -17830.482} C_VEL
LIN {X 0,Y 270.369,Z 162.409,A -85,B 0,C 180,E1 -17835.067,E2 -17835.067} C_VEL
LIN {X 0,Y 270.224,Z 162.428,A -85,B 0,C 180,E1 -17839.762,E2 -17839.762} C_VEL
LIN {X 0,Y 270.183,Z 162.438,A -85,B 0,C 180,E1 -17844.436,E2 -17844.436} C_VEL
LIN {X 0,Y 270.198,Z 162.453,A -85,B 0,C 180,E1 -17847.917,E2 -17847.917} C_VEL
LIN {X 0,Y 270.174,Z 162.389,A -85,B 0,C 180,E1 -17851.35,E2 -17851.35} C_VEL
LIN {X 0,Y 270.199,Z 162.42,A -85,B 0,C 180,E1 -17854.906,E2 -17854.906} C_VEL
LIN {X 0,Y 270.168,Z 162.413,A -85,B 0,C 180,E1 -17858.702,E2 -17858.702} C_VEL
LIN {X 0,Y 270.149,Z 162.454,A -85,B 0,C 180,E1 -17863.245,E2 -17863.245} C_VEL
LIN {X 0,Y 270.163,Z 162.786,A -85,B 0,C 180,E1 -17864.24,E2 -17864.24} C_VEL
LIN {X 0,Y 270.586,Z 164.148,A -85,B 0,C 180,E1 -17864.688,E2 -17864.688} C_VEL
LIN {X 0,Y 273.599,Z 168.611,A -85,B 0,C 180,E1 -17865.515,E2 -17865.515} C_VEL
LIN {X 0,Y 280.484,Z 179.649,A -85,B 0,C 180,E1 -17867.264,E2 -17867.264} C_VEL
LIN {X 0,Y 288.656,Z 193.726,A -85,B 0,C 180,E1 -17869.205,E2 -17869.205} C_VEL
LIN {X 0,Y 296.229,Z 208.782,A -85,B 0,C 180,E1 -17870.924,E2 -17870.924} C_VEL
LIN {X 0,Y 302.681,Z 223.31,A -85,B 0,C 180,E1 -17872.34,E2 -17872.34} C_VEL
LIN {X 0,Y 298.122,Z 329.054,A -85,B 0,C 180,E1 -17874.824,E2 -17874.824} C_VEL
LIN {X 0,Y 296.729,Z 344.251,A -85,B 0,C 180,E1 -17875.41,E2 -17875.41} C_VEL
LIN {X 0,Y 294.883,Z 359.018,A -85,B 0,C 180,E1 -17876.247,E2 -17876.247} C_VEL
LIN {X 0,Y 292.682,Z 373.136,A -85,B 0,C 180,E1 -17877.325,E2 -17877.325} C_VEL
LIN {X 0,Y 289.852,Z 388.006,A -85,B 0,C 180,E1 -17878.783,E2 -17878.783} C_VEL
LIN {X 0,Y 286.723,Z 401.491,A -85,B 0,C 180,E1 -17880.443,E2 -17880.443} C_VEL
LIN {X 0,Y 283.651,Z 413.73,A -85,B 0,C 180,E1 -17882.318,E2 -17882.318} C_VEL
LIN {X 0,Y 280.806,Z 424.302,A -85,B 0,C 180,E1 -17884.291,E2 -17884.291} C_VEL
LIN {X 0,Y 278.062,Z 434.262,A -85,B 0,C 180,E1 -17886.542,E2 -17886.542} C_VEL
LIN {X 0,Y 275.358,Z 443.488,A -85,B 0,C 180,E1 -17889.064,E2 -17889.064} C_VEL
LIN {X 0,Y 273.119,Z 451.159,A -85,B 0,C 180,E1 -17891.626,E2 -17891.626} C_VEL
LIN {X 0,Y 271.38,Z 457.524,A -85,B 0,C 180,E1 -17894.221,E2 -17894.221} C_VEL
LIN {X 0,Y 269.89,Z 463.371,A -85,B 0,C 180,E1 -17897.212,E2 -17897.212} C_VEL
LIN {X 0,Y 269.169,Z 466.833,A -85,B 0,C 180,E1 -17899.469,E2 -17899.469} C_VEL
LIN {X 0,Y 268.479,Z 470.341,A -85,B 0,C 180,E1 -17902.479,E2 -17902.479} C_VEL
LIN {X 0,Y 268.192,Z 472.658,A -85,B 0,C 180,E1 -17905.491,E2 -17905.491} C_VEL
LIN {X 0,Y 268.14,Z 473.839,A -85,B 0,C 180,E1 -17908.498,E2 -17908.498} C_VEL
LIN {X 0,Y 268.14,Z 473.853,A -85,B 0,C 180,E1 -17911.502,E2 -17911.502} C_VEL
LIN {X 0,Y 268.183,Z 472.726,A -85,B 0,C 180,E1 -17914.509,E2 -17914.509} C_VEL
LIN {X 0,Y 268.446,Z 470.461,A -85,B 0,C 180,E1 -17917.522,E2 -17917.522} C_VEL
LIN {X 0,Y 269.142,Z 467.001,A -85,B 0,C 180,E1 -17920.532,E2 -17920.532} C_VEL
LIN {X 0,Y 270.222,Z 462.266,A -85,B 0,C 180,E1 -17923.537,E2 -17923.537} C_VEL
LIN {X 0,Y 271.784,Z 456.134,A -85,B 0,C 180,E1 -17926.526,E2 -17926.526} C_VEL
LIN {X 0,Y 273.96,Z 448.412,A -85,B 0,C 180,E1 -17929.481,E2 -17929.481} C_VEL
LIN {X 0,Y 276.335,Z 440.182,A -85,B 0,C 180,E1 -17932.033,E2 -17932.033} C_VEL
LIN {X 0,Y 279.327,Z 430.267,A -85,B 0,C 180,E1 -17934.529,E2 -17934.529} C_VEL
LIN {X 0,Y 281.542,Z 421.879,A -85,B 0,C 180,E1 -17936.302,E2 -17936.302} C_VEL
LIN {X 0,Y 284.683,Z 410.142,A -85,B 0,C 180,E1 -17938.374,E2 -17938.374} C_VEL
LIN {X 0,Y 287.557,Z 398.452,A -85,B 0,C 180,E1 -17940.068,E2 -17940.068} C_VEL
LIN {X 0,Y 290.309,Z 385.85,A -85,B 0,C 180,E1 -17941.568,E2 -17941.568} C_VEL
LIN {X 0,Y 292.897,Z 372.469,A -85,B 0,C 180,E1 -17942.843,E2 -17942.843} C_VEL
LIN {X 0,Y 295.057,Z 358.011,A -85,B 0,C 180,E1 -17943.936,E2 -17943.936} C_VEL
LIN {X 0,Y 296.966,Z 342.847,A -85,B 0,C 180,E1 -17944.765,E2 -17944.765} C_VEL
LIN {X 0,Y 298.238,Z 328.318,A -85,B 0,C 180,E1 -17945.316,E2 -17945.316} C_VEL
LIN {X 0,Y 302.747,Z 224.542,A -85,B 0,C 180,E1 -17947.742,E2 -17947.742} C_VEL
LIN {X 0,Y 302.524,Z 222.767,A -85,B 0,C 180,E1 -17947.827,E2 -17947.827} C_VEL
LIN {X 0,Y 294.864,Z 205.742,A -85,B 0,C 180,E1 -17949.519,E2 -17949.519} C_VEL
LIN {X 0,Y 286.815,Z 190.353,A -85,B 0,C 180,E1 -17951.362,E2 -17951.362} C_VEL
LIN {X 0,Y 278.644,Z 176.601,A -85,B 0,C 180,E1 -17953.336,E2 -17953.336} C_VEL
LIN {X 0,Y 273.079,Z 167.944,A -85,B 0,C 180,E1 -17954.763,E2 -17954.763} C_VEL
LIN {X 0,Y 270.437,Z 163.833,A -85,B 0,C 180,E1 -17955.534,E2 -17955.534} C_VEL
LIN {X 0,Y 270.136,Z 162.594,A -85,B 0,C 180,E1 -17956.036,E2 -17956.036} C_VEL
LIN {X 0,Y 270.129,Z 162.409,A -85,B 0,C 180,E1 -17959.426,E2 -17959.426} C_VEL
LIN {X 0,Y 270.138,Z 162.427,A -85,B 0,C 180,E1 -17962.066,E2 -17962.066} C_VEL
LIN {X 0,Y 269.477,Z 162.542,A -85,B 0,C 180,E1 -17963.311,E2 -17963.311} C_VEL
LIN {X 0,Y 266.615,Z 162.862,A -85,B 0,C 180,E1 -17965.339,E2 -17965.339} C_VEL
LIN {X 0,Y 264.201,Z 163.138,A -85,B 0,C 180,E1 -17966.987,E2 -17966.987} C_VEL
LIN {X 0,Y 263.195,Z 163.255,A -85,B 0,C 180,E1 -17968.266,E2 -17968.266} C_VEL
LIN {X 0,Y 263.129,Z 163.265,A -85,B 0,C 180,E1 -17968.699,E2 -17968.699} C_VEL
LIN {X 0,Y 263.139,Z 163.33,A -85,B 0,C 180,E1 -17972.997,E2 -17972.997} C_VEL
LIN {X 0,Y 263.118,Z 163.325,A -85,B 0,C 180,E1 -17976.381,E2 -17976.381} C_VEL
LIN {X 0,Y 263.21,Z 163.301,A -85,B 0,C 180,E1 -17979.689,E2 -17979.689} C_VEL
LIN {X 0,Y 263.311,Z 163.292,A -85,B 0,C 180,E1 -17984.519,E2 -17984.519} C_VEL
LIN {X 0,Y 263.351,Z 163.303,A -85,B 0,C 180,E1 -17989.233,E2 -17989.233} C_VEL
LIN {X 0,Y 263.53,Z 163.261,A -85,B 0,C 180,E1 -17992.337,E2 -17992.337} C_VEL
LIN {X 0,Y 263.742,Z 163.233,A -85,B 0,C 180,E1 -17998.473,E2 -17998.473} C_VEL
LIN {X 0,Y 263.747,Z 163.247,A -85,B 0,C 180,E1 -18001.527,E2 -18001.527} C_VEL
LIN {X 0,Y 263.53,Z 163.276,A -85,B 0,C 180,E1 -18007.663,E2 -18007.663} C_VEL
LIN {X 0,Y 263.355,Z 163.286,A -85,B 0,C 180,E1 -18010.766,E2 -18010.766} C_VEL
LIN {X 0,Y 263.352,Z 163.282,A -85,B 0,C 180,E1 -18015.478,E2 -18015.478} C_VEL
LIN {X 0,Y 263.264,Z 163.297,A -85,B 0,C 180,E1 -18020.306,E2 -18020.306} C_VEL
LIN {X 0,Y 263.193,Z 163.308,A -85,B 0,C 180,E1 -18025.293,E2 -18025.293} C_VEL
LIN {X 0,Y 263.181,Z 163.327,A -85,B 0,C 180,E1 -18028.729,E2 -18028.729} C_VEL
LIN {X 0,Y 263.134,Z 163.265,A -85,B 0,C 180,E1 -18032.288,E2 -18032.288} C_VEL
LIN {X 0,Y 263.182,Z 163.327,A -85,B 0,C 180,E1 -18036.763,E2 -18036.763} C_VEL
LIN {X 0,Y 263.131,Z 163.416,A -85,B 0,C 180,E1 -18041.46,E2 -18041.46} C_VEL
LIN {X 0,Y 264.309,Z 167.173,A -85,B 0,C 180,E1 -18043.146,E2 -18043.146} C_VEL
LIN {X 0,Y 268.753,Z 174.256,A -85,B 0,C 180,E1 -18044.463,E2 -18044.463} C_VEL
LIN {X 0,Y 272.069,Z 179.418,A -85,B 0,C 180,E1 -18045.357,E2 -18045.357} C_VEL
LIN {X 0,Y 277.927,Z 189.214,A -85,B 0,C 180,E1 -18046.876,E2 -18046.876} C_VEL
LIN {X 0,Y 284.18,Z 200.584,A -85,B 0,C 180,E1 -18048.421,E2 -18048.421} C_VEL
LIN {X 0,Y 291.941,Z 216.421,A -85,B 0,C 180,E1 -18050.254,E2 -18050.254} C_VEL
LIN {X 0,Y 296.995,Z 228.216,A -85,B 0,C 180,E1 -18051.417,E2 -18051.417} C_VEL
LIN {X 0,Y 292.871,Z 321.86,A -85,B 0,C 180,E1 -18053.617,E2 -18053.617} C_VEL
LIN {X 0,Y 291.856,Z 338.782,A -85,B 0,C 180,E1 -18054.112,E2 -18054.112} C_VEL
LIN {X 0,Y 290.234,Z 353.778,A -85,B 0,C 180,E1 -18054.787,E2 -18054.787} C_VEL
LIN {X 0,Y 288.073,Z 367.852,A -85,B 0,C 180,E1 -18055.655,E2 -18055.655} C_VEL
LIN {X 0,Y 285.52,Z 382.649,A -85,B 0,C 180,E1 -18056.898,E2 -18056.898} C_VEL
LIN {X 0,Y 282.708,Z 395.996,A -85,B 0,C 180,E1 -18058.321,E2 -18058.321} C_VEL
LIN {X 0,Y 279.492,Z 408.888,A -85,B 0,C 180,E1 -18060.015,E2 -18060.015} C_VEL
LIN {X 0,Y 276.289,Z 420.693,A -85,B 0,C 180,E1 -18061.927,E2 -18061.927} C_VEL
LIN {X 0,Y 273.245,Z 431.509,A -85,B 0,C 180,E1 -18064.071,E2 -18064.071} C_VEL
LIN {X 0,Y 270.603,Z 440.685,A -85,B 0,C 180,E1 -18066.262,E2 -18066.262} C_VEL
LIN {X 0,Y 267.818,Z 449.684,A -85,B 0,C 180,E1 -18068.849,E2 -18068.849} C_VEL
LIN {X 0,Y 265.56,Z 457.149,A -85,B 0,C 180,E1 -18071.483,E2 -18071.483} C_VEL
LIN {X 0,Y 263.704,Z 464.113,A -85,B 0,C 180,E1 -18074.543,E2 -18074.543} C_VEL
LIN {X 0,Y 262.296,Z 469.586,A -85,B 0,C 180,E1 -18077.622,E2 -18077.622} C_VEL
LIN {X 0,Y 261.524,Z 473.725,A -85,B 0,C 180,E1 -18080.721,E2 -18080.721} C_VEL
LIN {X 0,Y 261.136,Z 476.625,A -85,B 0,C 180,E1 -18083.82,E2 -18083.82} C_VEL
LIN {X 0,Y 260.997,Z 478.353,A -85,B 0,C 180,E1 -18086.913,E2 -18086.913} C_VEL
LIN {X 0,Y 261.071,Z 478.944,A -85,B 0,C 180,E1 -18090,E2 -18090} C_VEL
LIN {X 0,Y 260.997,Z 478.341,A -85,B 0,C 180,E1 -18093.087,E2 -18093.087} C_VEL
LIN {X 0,Y 261.135,Z 476.597,A -85,B 0,C 180,E1 -18096.18,E2 -18096.18} C_VEL
LIN {X 0,Y 261.522,Z 473.685,A -85,B 0,C 180,E1 -18099.279,E2 -18099.279} C_VEL
LIN {X 0,Y 262.291,Z 469.538,A -85,B 0,C 180,E1 -18102.378,E2 -18102.378} C_VEL
LIN {X 0,Y 263.668,Z 464.046,A -85,B 0,C 180,E1 -18105.459,E2 -18105.459} C_VEL
LIN {X 0,Y 265.559,Z 457.057,A -85,B 0,C 180,E1 -18108.517,E2 -18108.517} C_VEL
LIN {X 0,Y 267.791,Z 449.582,A -85,B 0,C 180,E1 -18111.153,E2 -18111.153} C_VEL
LIN {X 0,Y 270.604,Z 440.568,A -85,B 0,C 180,E1 -18113.738,E2 -18113.738} C_VEL
LIN {X 0,Y 273.157,Z 431.365,A -85,B 0,C 180,E1 -18115.937,E2 -18115.937} C_VEL
LIN {X 0,Y 276.333,Z 420.524,A -85,B 0,C 180,E1 -18118.068,E2 -18118.068} C_VEL
LIN {X 0,Y 279.471,Z 408.688,A -85,B 0,C 180,E1 -18119.987,E2 -18119.987} C_VEL
LIN {X 0,Y 282.665,Z 395.741,A -85,B 0,C 180,E1 -18121.684,E2 -18121.684} C_VEL
LIN {X 0,Y 285.599,Z 382.018,A -85,B 0,C 180,E1 -18123.127,E2 -18123.127} C_VEL
LIN {X 0,Y 288.049,Z 367.445,A -85,B 0,C 180,E1 -18124.348,E2 -18124.348} C_VEL
LIN {X 0,Y 290.264,Z 352.476,A -85,B 0,C 180,E1 -18125.262,E2 -18125.262} C_VEL
LIN {X 0,Y 291.901,Z 336.814,A -85,B 0,C 180,E1 -18125.935,E2 -18125.935} C_VEL
LIN {X 0,Y 293.014,Z 316.964,A -85,B 0,C 180,E1 -18126.469,E2 -18126.469} C_VEL
LIN {X 0,Y 296.904,Z 228.062,A -85,B 0,C 180,E1 -18128.561,E2 -18128.561} C_VEL
LIN {X 0,Y 289.585,Z 211.447,A -85,B 0,C 180,E1 -18130.247,E2 -18130.247} C_VEL
LIN {X 0,Y 281.114,Z 194.778,A -85,B 0,C 180,E1 -18132.281,E2 -18132.281} C_VEL
LIN {X 0,Y 273.183,Z 181.163,A -85,B 0,C 180,E1 -18134.294,E2 -18134.294} C_VEL
LIN {X 0,Y 266.758,Z 171.195,A -85,B 0,C 180,E1 -18136.029,E2 -18136.029} C_VEL
LIN {X 0,Y 264.244,Z 166.978,A -85,B 0,C 180,E1 -18136.841,E2 -18136.841} C_VEL
LIN {X 0,Y 263.133,Z 163.426,A -85,B 0,C 180,E1 -18138.469,E2 -18138.469} C_VEL
LIN {X 0,Y 263.166,Z 163.315,A -85,B 0,C 180,E1 -18142.104,E2 -18142.104} C_VEL
LIN {X 0,Y 263.184,Z 163.263,A -85,B 0,C 180,E1 -18145.891,E2 -18145.891} C_VEL
LIN {X 0,Y 263.151,Z 163.292,A -85,B 0,C 180,E1 -18149.507,E2 -18149.507} C_VEL
LIN {X 0,Y 263.195,Z 163.309,A -85,B 0,C 180,E1 -18153.003,E2 -18153.003} C_VEL
LIN {X 0,Y 263.19,Z 163.326,A -85,B 0,C 180,E1 -18156.388,E2 -18156.388} C_VEL
LIN {X 0,Y 263.265,Z 163.297,A -85,B 0,C 180,E1 -18159.694,E2 -18159.694} C_VEL
LIN {X 0,Y 263.352,Z 163.282,A -85,B 0,C 180,E1 -18164.522,E2 -18164.522} C_VEL
LIN {X 0,Y 263.354,Z 163.285,A -85,B 0,C 180,E1 -18169.234,E2 -18169.234} C_VEL
LIN {X 0,Y 263.529,Z 163.276,A -85,B 0,C 180,E1 -18172.337,E2 -18172.337} C_VEL
LIN {X 0,Y 263.749,Z 163.247,A -85,B 0,C 180,E1 -18178.473,E2 -18178.473} C_VEL
LIN {X 0,Y 263.742,Z 163.233,A -85,B 0,C 180,E1 -18181.527,E2 -18181.527} C_VEL
LIN {X 0,Y 263.53,Z 163.261,A -85,B 0,C 180,E1 -18187.663,E2 -18187.663} C_VEL
LIN {X 0,Y 263.354,Z 163.301,A -85,B 0,C 180,E1 -18190.767,E2 -18190.767} C_VEL
LIN {X 0,Y 263.311,Z 163.291,A -85,B 0,C 180,E1 -18195.481,E2 -18195.481} C_VEL
LIN {X 0,Y 263.21,Z 163.301,A -85,B 0,C 180,E1 -18200.311,E2 -18200.311} C_VEL
LIN {X 0,Y 263.127,Z 163.313,A -85,B 0,C 180,E1 -18205.3,E2 -18205.3} C_VEL
LIN {X 0,Y 263.13,Z 163.321,A -85,B 0,C 180,E1 -18208.736,E2 -18208.736} C_VEL
LIN {X 0,Y 263.128,Z 163.262,A -85,B 0,C 180,E1 -18212.289,E2 -18212.289} C_VEL
LIN {X 0,Y 263.157,Z 163.328,A -85,B 0,C 180,E1 -18215.983,E2 -18215.983} C_VEL
LIN {X 0,Y 263.072,Z 163.285,A -85,B 0,C 180,E1 -18219.879,E2 -18219.879} C_VEL
LIN {X 0,Y 263.14,Z 163.524,A -85,B 0,C 180,E1 -18222.731,E2 -18222.731} C_VEL
LIN {X 0,Y 263.351,Z 164.494,A -85,B 0,C 180,E1 -18223.079,E2 -18223.079} C_VEL
LIN {X 0,Y 264.835,Z 167.19,A -85,B 0,C 180,E1 -18223.561,E2 -18223.561} C_VEL
LIN {X 0,Y 266.546,Z 169.124,A -85,B 0,C 180,E1 -18224.021,E2 -18224.021} C_VEL
LIN {X 0,Y 273.055,Z 179.008,A -85,B 0,C 180,E1 -18225.778,E2 -18225.778} C_VEL
LIN {X 0,Y 281.595,Z 193.618,A -85,B 0,C 180,E1 -18227.945,E2 -18227.945} C_VEL
LIN {X 0,Y 288.171,Z 206.041,A -85,B 0,C 180,E1 -18229.518,E2 -18229.518} C_VEL
LIN {X 0,Y 296.113,Z 223.214,A -85,B 0,C 180,E1 -18231.346,E2 -18231.346} C_VEL
LIN {X 0,Y 296.99,Z 225.363,A -85,B 0,C 180,E1 -18231.547,E2 -18231.547} C_VEL
LIN {X 0,Y 292.441,Z 327.727,A -85,B 0,C 180,E1 -18233.982,E2 -18233.982} C_VEL
LIN {X 0,Y 291.012,Z 343.442,A -85,B 0,C 180,E1 -18234.577,E2 -18234.577} C_VEL
LIN {X 0,Y 289.004,Z 359.093,A -85,B 0,C 180,E1 -18235.465,E2 -18235.465} C_VEL
LIN {X 0,Y 286.576,Z 374.065,A -85,B 0,C 180,E1 -18236.632,E2 -18236.632} C_VEL
LIN {X 0,Y 283.794,Z 388.078,A -85,B 0,C 180,E1 -18238.039,E2 -18238.039} C_VEL
LIN {X 0,Y 280.544,Z 401.562,A -85,B 0,C 180,E1 -18239.724,E2 -18239.724} C_VEL
LIN {X 0,Y 277.383,Z 413.8,A -85,B 0,C 180,E1 -18241.636,E2 -18241.636} C_VEL
LIN {X 0,Y 274.201,Z 425.025,A -85,B 0,C 180,E1 -18243.777,E2 -18243.777} C_VEL
LIN {X 0,Y 271.064,Z 435.784,A -85,B 0,C 180,E1 -18246.305,E2 -18246.305} C_VEL
LIN {X 0,Y 268.316,Z 444.778,A -85,B 0,C 180,E1 -18248.89,E2 -18248.89} C_VEL
LIN {X 0,Y 266.04,Z 452.232,A -85,B 0,C 180,E1 -18251.518,E2 -18251.518} C_VEL
LIN {X 0,Y 264.117,Z 459.2,A -85,B 0,C 180,E1 -18254.568,E2 -18254.568} C_VEL
LIN {X 0,Y 262.601,Z 464.676,A -85,B 0,C 180,E1 -18257.637,E2 -18257.637} C_VEL
LIN {X 0,Y 261.722,Z 468.808,A -85,B 0,C 180,E1 -18260.728,E2 -18260.728} C_VEL
LIN {X 0,Y 261.233,Z 471.711,A -85,B 0,C 180,E1 -18263.822,E2 -18263.822} C_VEL
LIN {X 0,Y 261.068,Z 473.455,A -85,B 0,C 180,E1 -18266.914,E2 -18266.914} C_VEL
LIN {X 0,Y 261.074,Z 474.063,A -85,B 0,C 180,E1 -18270,E2 -18270} C_VEL
LIN {X 0,Y 261.066,Z 473.495,A -85,B 0,C 180,E1 -18273.086,E2 -18273.086} C_VEL
LIN {X 0,Y 261.227,Z 471.804,A -85,B 0,C 180,E1 -18276.178,E2 -18276.178} C_VEL
LIN {X 0,Y 261.709,Z 468.95,A -85,B 0,C 180,E1 -18279.272,E2 -18279.272} C_VEL
LIN {X 0,Y 262.573,Z 464.866,A -85,B 0,C 180,E1 -18282.364,E2 -18282.364} C_VEL
LIN {X 0,Y 264.08,Z 459.45,A -85,B 0,C 180,E1 -18285.434,E2 -18285.434} C_VEL
LIN {X 0,Y 265.992,Z 452.552,A -85,B 0,C 180,E1 -18288.485,E2 -18288.485} C_VEL
LIN {X 0,Y 268.583,Z 443.942,A -85,B 0,C 180,E1 -18291.49,E2 -18291.49} C_VEL
LIN {X 0,Y 271.499,Z 434.788,A -85,B 0,C 180,E1 -18294.061,E2 -18294.061} C_VEL
LIN {X 0,Y 274.522,Z 424.085,A -85,B 0,C 180,E1 -18296.535,E2 -18296.535} C_VEL
LIN {X 0,Y 277.871,Z 412.34,A -85,B 0,C 180,E1 -18298.722,E2 -18298.722} C_VEL
LIN {X 0,Y 280.794,Z 401.084,A -85,B 0,C 180,E1 -18300.454,E2 -18300.454} C_VEL
LIN {X 0,Y 283.973,Z 387.49,A -85,B 0,C 180,E1 -18302.148,E2 -18302.148} C_VEL
LIN {X 0,Y 286.691,Z 373.996,A -85,B 0,C 180,E1 -18303.49,E2 -18303.49} C_VEL
LIN {X 0,Y 289.018,Z 359.35,A -85,B 0,C 180,E1 -18304.639,E2 -18304.639} C_VEL
LIN {X 0,Y 291.084,Z 343.815,A -85,B 0,C 180,E1 -18305.519,E2 -18305.519} C_VEL
LIN {X 0,Y 292.49,Z 328.364,A -85,B 0,C 180,E1 -18306.117,E2 -18306.117} C_VEL
LIN {X 0,Y 297.116,Z 226.14,A -85,B 0,C 180,E1 -18308.541,E2 -18308.541} C_VEL
LIN {X 0,Y 296.395,Z 223.868,A -85,B 0,C 180,E1 -18308.721,E2 -18308.721} C_VEL
LIN {X 0,Y 289.343,Z 208.358,A -85,B 0,C 180,E1 -18310.344,E2 -18310.344} C_VEL
LIN {X 0,Y 281.677,Z 193.668,A -85,B 0,C 180,E1 -18312.178,E2 -18312.178} C_VEL
LIN {X 0,Y 272.428,Z 178,A -85,B 0,C 180,E1 -18314.534,E2 -18314.534} C_VEL
LIN {X 0,Y 268.009,Z 171.458,A -85,B 0,C 180,E1 -18315.718,E2 -18315.718} C_VEL
LIN {X 0,Y 265.719,Z 168.062,A -85,B 0,C 180,E1 -18316.358,E2 -18316.358} C_VEL
LIN {X 0,Y 263.763,Z 165.534,A -85,B 0,C 180,E1 -18316.908,E2 -18316.908} C_VEL
LIN {X 0,Y 263.215,Z 163.925,A -85,B 0,C 180,E1 -18317.219,E2 -18317.219} C_VEL
LIN {X 0,Y 263.118,Z 163.397,A -85,B 0,C 180,E1 -18317.589,E2 -18317.589} C_VEL
LIN {X 0,Y 263.107,Z 163.302,A -85,B 0,C 180,E1 -18322.094,E2 -18322.094} C_VEL
LIN {X 0,Y 263.153,Z 163.28,A -85,B 0,C 180,E1 -18325.885,E2 -18325.885} C_VEL
LIN {X 0,Y 263.129,Z 163.265,A -85,B 0,C 180,E1 -18328.699,E2 -18328.699} C_VEL
LIN {X 0,Y 262.497,Z 163.367,A -85,B 0,C 180,E1 -18329.976,E2 -18329.976} C_VEL
LIN {X 0,Y 259.636,Z 163.768,A -85,B 0,C 180,E1 -18332.055,E2 -18332.055} C_VEL
LIN {X 0,Y 257.193,Z 164.063,A -85,B 0,C 180,E1 -18333.747,E2 -18333.747} C_VEL
LIN {X 0,Y 256.158,Z 164.182,A -85,B 0,C 180,E1 -18335.06,E2 -18335.06} C_VEL
LIN {X 0,Y 256.083,Z 164.192,A -85,B 0,C 180,E1 -18335.505,E2 -18335.505} C_VEL
LIN {X 0,Y 256.123,Z 164.187,A -85,B 0,C 180,E1 -18339.101,E2 -18339.101} C_VEL
LIN {X 0,Y 256.231,Z 164.179,A -85,B 0,C 180,E1 -18344.08,E2 -18344.08} C_VEL
LIN {X 0,Y 256.292,Z 164.185,A -85,B 0,C 180,E1 -18348.933,E2 -18348.933} C_VEL
LIN {X 0,Y 256.472,Z 164.138,A -85,B 0,C 180,E1 -18352.125,E2 -18352.125} C_VEL
LIN {X 0,Y 256.459,Z 164.138,A -85,B 0,C 180,E1 -18356.858,E2 -18356.858} C_VEL
LIN {X 0,Y 256.745,Z 164.123,A -85,B 0,C 180,E1 -18360,E2 -18360} C_VEL
LIN {X 0,Y 256.486,Z 164.133,A -85,B 0,C 180,E1 -18363.141,E2 -18363.141} C_VEL
LIN {X 0,Y 256.472,Z 164.151,A -85,B 0,C 180,E1 -18367.875,E2 -18367.875} C_VEL
LIN {X 0,Y 256.297,Z 164.168,A -85,B 0,C 180,E1 -18371.066,E2 -18371.066} C_VEL
LIN {X 0,Y 256.256,Z 164.172,A -85,B 0,C 180,E1 -18374.29,E2 -18374.29} C_VEL
LIN {X 0,Y 256.211,Z 164.19,A -85,B 0,C 180,E1 -18377.562,E2 -18377.562} C_VEL
LIN {X 0,Y 256.154,Z 164.18,A -85,B 0,C 180,E1 -18381.117,E2 -18381.117} C_VEL
LIN {X 0,Y 256.172,Z 164.184,A -85,B 0,C 180,E1 -18385.13,E2 -18385.13} C_VEL
LIN {X 0,Y 256.115,Z 164.189,A -85,B 0,C 180,E1 -18389.599,E2 -18389.599} C_VEL
LIN {X 0,Y 256.068,Z 164.142,A -85,B 0,C 180,E1 -18393.292,E2 -18393.292} C_VEL
LIN {X 0,Y 256.116,Z 164.206,A -85,B 0,C 180,E1 -18397.271,E2 -18397.271} C_VEL
LIN {X 0,Y 256.114,Z 164.379,A -85,B 0,C 180,E1 -18400.122,E2 -18400.122} C_VEL
LIN {X 0,Y 257.098,Z 167.259,A -85,B 0,C 180,E1 -18401.427,E2 -18401.427} C_VEL
LIN {X 0,Y 260.436,Z 172.312,A -85,B 0,C 180,E1 -18402.491,E2 -18402.491} C_VEL
LIN {X 0,Y 267.759,Z 183.888,A -85,B 0,C 180,E1 -18404.607,E2 -18404.607} C_VEL
LIN {X 0,Y 273.204,Z 192.987,A -85,B 0,C 180,E1 -18406.078,E2 -18406.078} C_VEL
LIN {X 0,Y 280.439,Z 206.433,A -85,B 0,C 180,E1 -18407.938,E2 -18407.938} C_VEL
LIN {X 0,Y 287.651,Z 221.603,A -85,B 0,C 180,E1 -18409.707,E2 -18409.707} C_VEL
LIN {X 0,Y 291.362,Z 230.387,A -85,B 0,C 180,E1 -18410.597,E2 -18410.597} C_VEL
LIN {X 0,Y 287.202,Z 321.816,A -85,B 0,C 180,E1 -18412.779,E2 -18412.779} C_VEL
LIN {X 0,Y 286.147,Z 338.729,A -85,B 0,C 180,E1 -18413.28,E2 -18413.28} C_VEL
LIN {X 0,Y 284.442,Z 353.72,A -85,B 0,C 180,E1 -18413.959,E2 -18413.959} C_VEL
LIN {X 0,Y 282.251,Z 367.792,A -85,B 0,C 180,E1 -18414.844,E2 -18414.844} C_VEL
LIN {X 0,Y 279.654,Z 382.279,A -85,B 0,C 180,E1 -18416.073,E2 -18416.073} C_VEL
LIN {X 0,Y 276.644,Z 395.933,A -85,B 0,C 180,E1 -18417.543,E2 -18417.543} C_VEL
LIN {X 0,Y 273.315,Z 408.825,A -85,B 0,C 180,E1 -18419.265,E2 -18419.265} C_VEL
LIN {X 0,Y 270.024,Z 420.629,A -85,B 0,C 180,E1 -18421.216,E2 -18421.216} C_VEL
LIN {X 0,Y 266.817,Z 431.445,A -85,B 0,C 180,E1 -18423.398,E2 -18423.398} C_VEL
LIN {X 0,Y 264.055,Z 440.62,A -85,B 0,C 180,E1 -18425.635,E2 -18425.635} C_VEL
LIN {X 0,Y 261.158,Z 449.619,A -85,B 0,C 180,E1 -18428.283,E2 -18428.283} C_VEL
LIN {X 0,Y 258.791,Z 457.084,A -85,B 0,C 180,E1 -18430.981,E2 -18430.981} C_VEL
LIN {X 0,Y 256.812,Z 464.047,A -85,B 0,C 180,E1 -18434.118,E2 -18434.118} C_VEL
LIN {X 0,Y 255.318,Z 469.52,A -85,B 0,C 180,E1 -18437.278,E2 -18437.278} C_VEL
LIN {X 0,Y 254.485,Z 473.659,A -85,B 0,C 180,E1 -18440.462,E2 -18440.462} C_VEL
LIN {X 0,Y 254.045,Z 476.559,A -85,B 0,C 180,E1 -18443.647,E2 -18443.647} C_VEL
LIN {X 0,Y 253.899,Z 478.287,A -85,B 0,C 180,E1 -18446.826,E2 -18446.826} C_VEL
LIN {X 0,Y 253.979,Z 478.878,A -85,B 0,C 180,E1 -18450,E2 -18450} C_VEL
LIN {X 0,Y 253.899,Z 478.275,A -85,B 0,C 180,E1 -18453.173,E2 -18453.173} C_VEL
LIN {X 0,Y 254.045,Z 476.53,A -85,B 0,C 180,E1 -18456.353,E2 -18456.353} C_VEL
LIN {X 0,Y 254.483,Z 473.618,A -85,B 0,C 180,E1 -18459.538,E2 -18459.538} C_VEL
LIN {X 0,Y 255.313,Z 469.47,A -85,B 0,C 180,E1 -18462.722,E2 -18462.722} C_VEL
LIN {X 0,Y 256.776,Z 463.977,A -85,B 0,C 180,E1 -18465.885,E2 -18465.885} C_VEL
LIN {X 0,Y 258.79,Z 456.989,A -85,B 0,C 180,E1 -18469.019,E2 -18469.019} C_VEL
LIN {X 0,Y 261.474,Z 448.293,A -85,B 0,C 180,E1 -18472.105,E2 -18472.105} C_VEL
LIN {X 0,Y 264.494,Z 439.055,A -85,B 0,C 180,E1 -18474.74,E2 -18474.74} C_VEL
LIN {X 0,Y 266.75,Z 431.296,A -85,B 0,C 180,E1 -18476.609,E2 -18476.609} C_VEL
LIN {X 0,Y 270.054,Z 420.455,A -85,B 0,C 180,E1 -18478.78,E2 -18478.78} C_VEL
LIN {X 0,Y 273.304,Z 408.618,A -85,B 0,C 180,E1 -18480.736,E2 -18480.736} C_VEL
LIN {X 0,Y 276.644,Z 395.67,A -85,B 0,C 180,E1 -18482.457,E2 -18482.457} C_VEL
LIN {X 0,Y 279.687,Z 381.819,A -85,B 0,C 180,E1 -18483.937,E2 -18483.937} C_VEL
LIN {X 0,Y 282.208,Z 367.372,A -85,B 0,C 180,E1 -18485.162,E2 -18485.162} C_VEL
LIN {X 0,Y 284.509,Z 352.401,A -85,B 0,C 180,E1 -18486.086,E2 -18486.086} C_VEL
LIN {X 0,Y 286.197,Z 336.734,A -85,B 0,C 180,E1 -18486.767,E2 -18486.767} C_VEL
LIN {X 0,Y 287.344,Z 316.876,A -85,B 0,C 180,E1 -18487.309,E2 -18487.309} C_VEL
LIN {X 0,Y 291.27,Z 230.172,A -85,B 0,C 180,E1 -18489.381,E2 -18489.381} C_VEL
LIN {X 0,Y 283.896,Z 213.467,A -85,B 0,C 180,E1 -18491.157,E2 -18491.157} C_VEL
LIN {X 0,Y 276.209,Z 198.44,A -85,B 0,C 180,E1 -18493.082,E2 -18493.082} C_VEL
LIN {X 0,Y 268.434,Z 184.938,A -85,B 0,C 180,E1 -18495.149,E2 -18495.149} C_VEL
LIN {X 0,Y 262.518,Z 175.745,A -85,B 0,C 180,E1 -18496.816,E2 -18496.816} C_VEL
LIN {X 0,Y 259.021,Z 170.438,A -85,B 0,C 180,E1 -18497.858,E2 -18497.858} C_VEL
LIN {X 0,Y 256.942,Z 166.871,A -85,B 0,C 180,E1 -18498.612,E2 -18498.612} C_VEL
LIN {X 0,Y 256.114,Z 164.296,A -85,B 0,C 180,E1 -18499.874,E2 -18499.874} C_VEL
LIN {X 0,Y 256.145,Z 164.205,A -85,B 0,C 180,E1 -18502.87,E2 -18502.87} C_VEL
LIN {X 0,Y 256.086,Z 164.14,A -85,B 0,C 180,E1 -18506.71,E2 -18506.71} C_VEL
LIN {X 0,Y 256.139,Z 164.206,A -85,B 0,C 180,E1 -18511.405,E2 -18511.405} C_VEL
LIN {X 0,Y 256.171,Z 164.196,A -85,B 0,C 180,E1 -18515.7,E2 -18515.7} C_VEL
LIN {X 0,Y 256.168,Z 164.178,A -85,B 0,C 180,E1 -18519.105,E2 -18519.105} C_VEL
LIN {X 0,Y 256.301,Z 164.16,A -85,B 0,C 180,E1 -18524.085,E2 -18524.085} C_VEL
LIN {X 0,Y 256.295,Z 164.186,A -85,B 0,C 180,E1 -18527.328,E2 -18527.328} C_VEL
LIN {X 0,Y 256.435,Z 164.141,A -85,B 0,C 180,E1 -18530.623,E2 -18530.623} C_VEL
LIN {X 0,Y 256.461,Z 164.162,A -85,B 0,C 180,E1 -18533.707,E2 -18533.707} C_VEL
LIN {X 0,Y 256.712,Z 164.123,A -85,B 0,C 180,E1 -18538.431,E2 -18538.431} C_VEL
LIN {X 0,Y 256.704,Z 164.108,A -85,B 0,C 180,E1 -18541.569,E2 -18541.569} C_VEL
LIN {X 0,Y 256.449,Z 164.155,A -85,B 0,C 180,E1 -18546.564,E2 -18546.564} C_VEL
LIN {X 0,Y 256.428,Z 164.146,A -85,B 0,C 180,E1 -18549.465,E2 -18549.465} C_VEL
LIN {X 0,Y 256.232,Z 164.167,A -85,B 0,C 180,E1 -18554.292,E2 -18554.292} C_VEL
LIN {X 0,Y 256.164,Z 164.201,A -85,B 0,C 180,E1 -18557.565,E2 -18557.565} C_VEL
LIN {X 0,Y 256.121,Z 164.189,A -85,B 0,C 180,E1 -18561.098,E2 -18561.098} C_VEL
LIN {X 0,Y 256.086,Z 164.19,A -85,B 0,C 180,E1 -18565.089,E2 -18565.089} C_VEL
LIN {X 0,Y 256.088,Z 164.201,A -85,B 0,C 180,E1 -18568.574,E2 -18568.574} C_VEL
LIN {X 0,Y 256.074,Z 164.14,A -85,B 0,C 180,E1 -18571.701,E2 -18571.701} C_VEL
LIN {X 0,Y 256.08,Z 164.181,A -85,B 0,C 180,E1 -18575.193,E2 -18575.193} C_VEL
LIN {X 0,Y 256.042,Z 164.164,A -85,B 0,C 180,E1 -18579.148,E2 -18579.148} C_VEL
LIN {X 0,Y 256.047,Z 164.365,A -85,B 0,C 180,E1 -18581.007,E2 -18581.007} C_VEL
LIN {X 0,Y 256.305,Z 165.432,A -85,B 0,C 180,E1 -18581.416,E2 -18581.416} C_VEL
LIN {X 0,Y 257.905,Z 168.147,A -85,B 0,C 180,E1 -18581.951,E2 -18581.951} C_VEL
LIN {X 0,Y 259.501,Z 169.764,A -85,B 0,C 180,E1 -18582.408,E2 -18582.408} C_VEL
LIN {X 0,Y 261.739,Z 173.186,A -85,B 0,C 180,E1 -18583.079,E2 -18583.079} C_VEL
LIN {X 0,Y 263.118,Z 175.008,A -85,B 0,C 180,E1 -18583.471,E2 -18583.471} C_VEL
LIN {X 0,Y 267.292,Z 181.324,A -85,B 0,C 180,E1 -18584.647,E2 -18584.647} C_VEL
LIN {X 0,Y 274.495,Z 193.27,A -85,B 0,C 180,E1 -18586.577,E2 -18586.577} C_VEL
LIN {X 0,Y 281.822,Z 206.793,A -85,B 0,C 180,E1 -18588.429,E2 -18588.429} C_VEL
LIN {X 0,Y 288.213,Z 220.277,A -85,B 0,C 180,E1 -18589.981,E2 -18589.981} C_VEL
LIN {X 0,Y 291.368,Z 227.523,A -85,B 0,C 180,E1 -18590.728,E2 -18590.728} C_VEL
LIN {X 0,Y 286.652,Z 329.219,A -85,B 0,C 180,E1 -18593.191,E2 -18593.191} C_VEL
LIN {X 0,Y 285.093,Z 345.187,A -85,B 0,C 180,E1 -18593.836,E2 -18593.836} C_VEL
LIN {X 0,Y 282.996,Z 360.335,A -85,B 0,C 180,E1 -18594.732,E2 -18594.732} C_VEL
LIN {X 0,Y 280.525,Z 374.893,A -85,B 0,C 180,E1 -18595.906,E2 -18595.906} C_VEL
LIN {X 0,Y 277.773,Z 388.149,A -85,B 0,C 180,E1 -18597.261,E2 -18597.261} C_VEL
LIN {X 0,Y 274.443,Z 401.632,A -85,B 0,C 180,E1 -18598.978,E2 -18598.978} C_VEL
LIN {X 0,Y 271.149,Z 413.87,A -85,B 0,C 180,E1 -18600.923,E2 -18600.923} C_VEL
LIN {X 0,Y 267.782,Z 425.193,A -85,B 0,C 180,E1 -18603.124,E2 -18603.124} C_VEL
LIN {X 0,Y 264.559,Z 435.852,A -85,B 0,C 180,E1 -18605.685,E2 -18605.685} C_VEL
LIN {X 0,Y 261.661,Z 444.847,A -85,B 0,C 180,E1 -18608.327,E2 -18608.327} C_VEL
LIN {X 0,Y 258.938,Z 453.353,A -85,B 0,C 180,E1 -18611.438,E2 -18611.438} C_VEL
LIN {X 0,Y 257.204,Z 459.268,A -85,B 0,C 180,E1 -18614.142,E2 -18614.142} C_VEL
LIN {X 0,Y 255.626,Z 464.743,A -85,B 0,C 180,E1 -18617.294,E2 -18617.294} C_VEL
LIN {X 0,Y 254.704,Z 468.875,A -85,B 0,C 180,E1 -18620.47,E2 -18620.47} C_VEL
LIN {X 0,Y 254.16,Z 471.778,A -85,B 0,C 180,E1 -18623.65,E2 -18623.65} C_VEL
LIN {X 0,Y 253.969,Z 473.522,A -85,B 0,C 180,E1 -18626.827,E2 -18626.827} C_VEL
LIN {X 0,Y 253.982,Z 474.129,A -85,B 0,C 180,E1 -18630,E2 -18630} C_VEL
LIN {X 0,Y 253.966,Z 473.562,A -85,B 0,C 180,E1 -18633.173,E2 -18633.173} C_VEL
LIN {X 0,Y 254.155,Z 471.87,A -85,B 0,C 180,E1 -18636.351,E2 -18636.351} C_VEL
LIN {X 0,Y 254.688,Z 469.016,A -85,B 0,C 180,E1 -18639.53,E2 -18639.53} C_VEL
LIN {X 0,Y 255.6,Z 464.931,A -85,B 0,C 180,E1 -18642.707,E2 -18642.707} C_VEL
LIN {X 0,Y 257.165,Z 459.516,A -85,B 0,C 180,E1 -18645.86,E2 -18645.86} C_VEL
LIN {X 0,Y 259.236,Z 452.617,A -85,B 0,C 180,E1 -18648.985,E2 -18648.985} C_VEL
LIN {X 0,Y 261.96,Z 444.006,A -85,B 0,C 180,E1 -18652.062,E2 -18652.062} C_VEL
LIN {X 0,Y 264.991,Z 434.852,A -85,B 0,C 180,E1 -18654.691,E2 -18654.691} C_VEL
LIN {X 0,Y 267.683,Z 425.695,A -85,B 0,C 180,E1 -18656.887,E2 -18656.887} C_VEL
LIN {X 0,Y 271.345,Z 413.467,A -85,B 0,C 180,E1 -18659.267,E2 -18659.267} C_VEL
LIN {X 0,Y 274.691,Z 401.146,A -85,B 0,C 180,E1 -18661.205,E2 -18661.205} C_VEL
LIN {X 0,Y 277.961,Z 387.551,A -85,B 0,C 180,E1 -18662.93,E2 -18662.93} C_VEL
LIN {X 0,Y 280.902,Z 373.419,A -85,B 0,C 180,E1 -18664.346,E2 -18664.346} C_VEL
LIN {X 0,Y 283.201,Z 359.408,A -85,B 0,C 180,E1 -18665.456,E2 -18665.456} C_VEL
LIN {X 0,Y 285.353,Z 343.869,A -85,B 0,C 180,E1 -18666.345,E2 -18666.345} C_VEL
LIN {X 0,Y 286.801,Z 328.41,A -85,B 0,C 180,E1 -18666.951,E2 -18666.951} C_VEL
LIN {X 0,Y 291.463,Z 228.728,A -85,B 0,C 180,E1 -18669.352,E2 -18669.352} C_VEL
LIN {X 0,Y 291.221,Z 227.064,A -85,B 0,C 180,E1 -18669.443,E2 -18669.443} C_VEL
LIN {X 0,Y 284.454,Z 212.111,A -85,B 0,C 180,E1 -18671.064,E2 -18671.064} C_VEL
LIN {X 0,Y 277.253,Z 198.165,A -85,B 0,C 180,E1 -18672.857,E2 -18672.857} C_VEL
LIN {X 0,Y 269.545,Z 184.854,A -85,B 0,C 180,E1 -18674.888,E2 -18674.888} C_VEL
LIN {X 0,Y 264.61,Z 177.141,A -85,B 0,C 180,E1 -18676.26,E2 -18676.26} C_VEL
LIN {X 0,Y 262.065,Z 173.504,A -85,B 0,C 180,E1 -18676.988,E2 -18676.988} C_VEL
LIN {X 0,Y 259.807,Z 170.323,A -85,B 0,C 180,E1 -18677.654,E2 -18677.654} C_VEL
LIN {X 0,Y 258.966,Z 169.12,A -85,B 0,C 180,E1 -18677.907,E2 -18677.907} C_VEL
LIN {X 0,Y 256.846,Z 166.72,A -85,B 0,C 180,E1 -18678.533,E2 -18678.533} C_VEL
LIN {X 0,Y 256.119,Z 164.826,A -85,B 0,C 180,E1 -18678.908,E2 -18678.908} C_VEL
LIN {X 0,Y 256.019,Z 164.242,A -85,B 0,C 180,E1 -18679.381,E2 -18679.381} C_VEL
LIN {X 0,Y 256.099,Z 164.192,A -85,B 0,C 180,E1 -18682.862,E2 -18682.862} C_VEL
LIN {X 0,Y 256.067,Z 164.147,A -85,B 0,C 180,E1 -18686.707,E2 -18686.707} C_VEL
LIN {X 0,Y 256.053,Z 164.171,A -85,B 0,C 180,E1 -18690.392,E2 -18690.392} C_VEL
LIN {X 0,Y 256.079,Z 164.195,A -85,B 0,C 180,E1 -18693.952,E2 -18693.952} C_VEL
LIN {X 0,Y 256.083,Z 164.192,A -85,B 0,C 180,E1 -18695.505,E2 -18695.505} C_VEL
LIN {X 0,Y 255.433,Z 164.289,A -85,B 0,C 180,E1 -18696.818,E2 -18696.818} C_VEL
LIN {X 0,Y 252.581,Z 164.64,A -85,B 0,C 180,E1 -18698.958,E2 -18698.958} C_VEL
LIN {X 0,Y 250.167,Z 164.94,A -85,B 0,C 180,E1 -18700.7,E2 -18700.7} C_VEL
LIN {X 0,Y 249.161,Z 165.068,A -85,B 0,C 180,E1 -18702.052,E2 -18702.052} C_VEL
LIN {X 0,Y 249.095,Z 165.071,A -85,B 0,C 180,E1 -18702.51,E2 -18702.51} C_VEL
LIN {X 0,Y 249.19,Z 165.053,A -85,B 0,C 180,E1 -18706.96,E2 -18706.96} C_VEL
LIN {X 0,Y 249.385,Z 165.023,A -85,B 0,C 180,E1 -18710.522,E2 -18710.522} C_VEL
LIN {X 0,Y 249.432,Z 165.031,A -85,B 0,C 180,E1 -18713.529,E2 -18713.529} C_VEL
LIN {X 0,Y 249.664,Z 164.984,A -85,B 0,C 180,E1 -18718.387,E2 -18718.387} C_VEL
LIN {X 0,Y 249.672,Z 164.999,A -85,B 0,C 180,E1 -18721.613,E2 -18721.613} C_VEL
LIN {X 0,Y 249.432,Z 165.038,A -85,B 0,C 180,E1 -18726.471,E2 -18726.471} C_VEL
LIN {X 0,Y 249.345,Z 165.023,A -85,B 0,C 180,E1 -18729.736,E2 -18729.736} C_VEL
LIN {X 0,Y 249.207,Z 165.046,A -85,B 0,C 180,E1 -18734.703,E2 -18734.703} C_VEL
LIN {X 0,Y 249.14,Z 165.076,A -85,B 0,C 180,E1 -18738.077,E2 -18738.077} C_VEL
LIN {X 0,Y 249.085,Z 165.061,A -85,B 0,C 180,E1 -18741.518,E2 -18741.518} C_VEL
LIN {X 0,Y 249.118,Z 165.06,A -85,B 0,C 180,E1 -18745.475,E2 -18745.475} C_VEL
LIN {X 0,Y 249.085,Z 165.079,A -85,B 0,C 180,E1 -18748.993,E2 -18748.993} C_VEL
LIN {X 0,Y 249.031,Z 165.018,A -85,B 0,C 180,E1 -18752.425,E2 -18752.425} C_VEL
LIN {X 0,Y 249.048,Z 165.07,A -85,B 0,C 180,E1 -18756.342,E2 -18756.342} C_VEL
LIN {X 0,Y 249.074,Z 165.344,A -85,B 0,C 180,E1 -18758.63,E2 -18758.63} C_VEL
LIN {X 0,Y 249.631,Z 167.126,A -85,B 0,C 180,E1 -18759.436,E2 -18759.436} C_VEL
LIN {X 0,Y 253.897,Z 173.446,A -85,B 0,C 180,E1 -18760.905,E2 -18760.905} C_VEL
LIN {X 0,Y 260.348,Z 183.196,A -85,B 0,C 180,E1 -18762.904,E2 -18762.904} C_VEL
LIN {X 0,Y 268.404,Z 196.549,A -85,B 0,C 180,E1 -18765.215,E2 -18765.215} C_VEL
LIN {X 0,Y 275.873,Z 210.618,A -85,B 0,C 180,E1 -18767.223,E2 -18767.223} C_VEL
LIN {X 0,Y 282.76,Z 225.293,A -85,B 0,C 180,E1 -18768.985,E2 -18768.985} C_VEL
LIN {X 0,Y 285.784,Z 232.426,A -85,B 0,C 180,E1 -18769.74,E2 -18769.74} C_VEL
LIN {X 0,Y 281.8,Z 318.193,A -85,B 0,C 180,E1 -18771.827,E2 -18771.827} C_VEL
LIN {X 0,Y 280.578,Z 337.537,A -85,B 0,C 180,E1 -18772.37,E2 -18772.37} C_VEL
LIN {X 0,Y 278.815,Z 352.901,A -85,B 0,C 180,E1 -18773.057,E2 -18773.057} C_VEL
LIN {X 0,Y 276.486,Z 367.733,A -85,B 0,C 180,E1 -18773.998,E2 -18773.998} C_VEL
LIN {X 0,Y 273.915,Z 381.641,A -85,B 0,C 180,E1 -18775.189,E2 -18775.189} C_VEL
LIN {X 0,Y 270.674,Z 395.871,A -85,B 0,C 180,E1 -18776.735,E2 -18776.735} C_VEL
LIN {X 0,Y 267.222,Z 408.762,A -85,B 0,C 180,E1 -18778.485,E2 -18778.485} C_VEL
LIN {X 0,Y 263.796,Z 420.565,A -85,B 0,C 180,E1 -18780.47,E2 -18780.47} C_VEL
LIN {X 0,Y 260.451,Z 431.38,A -85,B 0,C 180,E1 -18782.695,E2 -18782.695} C_VEL
LIN {X 0,Y 257.554,Z 440.555,A -85,B 0,C 180,E1 -18784.979,E2 -18784.979} C_VEL
LIN {X 0,Y 254.511,Z 449.554,A -85,B 0,C 180,E1 -18787.685,E2 -18787.685} C_VEL
LIN {X 0,Y 252.034,Z 457.019,A -85,B 0,C 180,E1 -18790.45,E2 -18790.45} C_VEL
LIN {X 0,Y 249.934,Z 463.981,A -85,B 0,C 180,E1 -18793.668,E2 -18793.668} C_VEL
